Yaskawa INFORM job: A_ROOF_SIDE_0617_2_PAINT_31.JBI

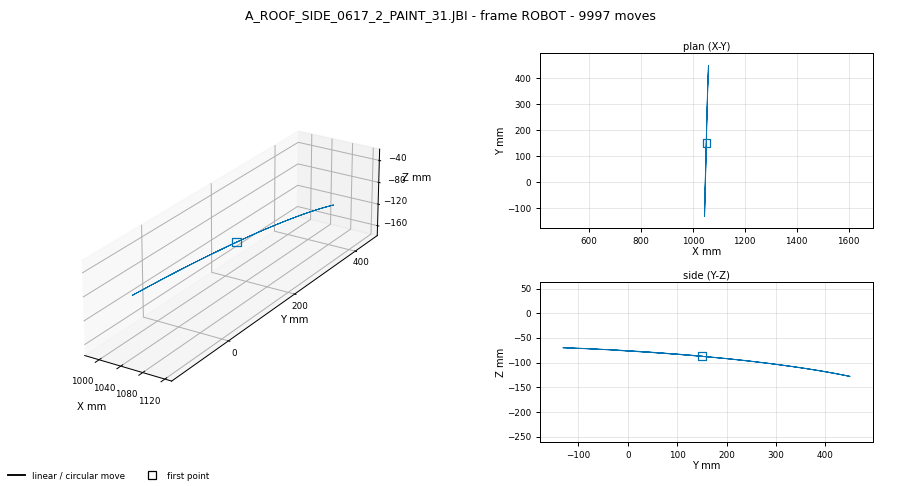
[picture p0: tool path of A_ROOF_SIDE_0617_2_PAINT_31.JBI in frame ROBOT, 9997 of 9997 moves have a stored position in this frame; points joined in program order, loops and branches not executed]
/JOB
//NAME A_ROOF_SIDE_0617_2_PAINT31
//POS
///NPOS 9997,0,0,0,0,0
///TOOL 1
///USER 0
///POSTYPE ROBOT
///RECTAN
///RCONF 1,0,0,0,0,0,0,0,0,0,0,0,0,0,0,0,0,0,0,0,0,0,0,0
C00000=1052.598,150.820,-86.690,171.369,34.301,156.430
C00001=1052.592,150.571,-86.668,171.366,34.299,156.430
C00002=1052.586,150.322,-86.647,171.364,34.297,156.430
C00003=1052.580,150.074,-86.625,171.362,34.294,156.429
C00004=1052.574,149.824,-86.603,171.360,34.291,156.429
C00005=1052.568,149.575,-86.581,171.358,34.290,156.428
C00006=1052.563,149.326,-86.560,171.357,34.287,156.428
C00007=1052.557,149.077,-86.538,171.355,34.285,156.427
C00008=1052.550,148.828,-86.516,171.353,34.283,156.427
C00009=1052.544,148.579,-86.494,171.351,34.280,156.427
C00010=1052.538,148.331,-86.473,171.349,34.278,156.426
C00011=1052.532,148.082,-86.451,171.347,34.276,156.426
C00012=1052.526,147.832,-86.429,171.345,34.273,156.425
C00013=1052.520,147.583,-86.408,171.343,34.271,156.425
C00014=1052.515,147.334,-86.386,171.341,34.269,156.425
C00015=1052.508,147.085,-86.365,171.339,34.267,156.424
C00016=1052.502,146.836,-86.343,171.337,34.264,156.424
C00017=1052.496,146.587,-86.322,171.335,34.262,156.424
C00018=1052.490,146.339,-86.300,171.334,34.260,156.423
C00019=1052.484,146.089,-86.279,171.332,34.258,156.423
C00020=1052.478,145.840,-86.257,171.330,34.255,156.422
C00021=1052.472,145.591,-86.236,171.328,34.253,156.422
C00022=1052.466,145.342,-86.214,171.326,34.251,156.422
C00023=1052.460,145.093,-86.193,171.324,34.248,156.421
C00024=1052.454,144.844,-86.171,171.322,34.246,156.421
C00025=1052.448,144.595,-86.150,171.320,34.244,156.420
C00026=1052.442,144.346,-86.128,171.318,34.242,156.420
C00027=1052.436,144.097,-86.106,171.316,34.239,156.420
C00028=1052.431,143.849,-86.085,171.314,34.237,156.419
C00029=1052.424,143.599,-86.064,171.313,34.235,156.419
C00030=1052.418,143.350,-86.042,171.311,34.233,156.418
C00031=1052.412,143.101,-86.020,171.309,34.230,156.418
C00032=1052.406,142.852,-85.999,171.307,34.228,156.418
C00033=1052.400,142.603,-85.979,171.305,34.226,156.417
C00034=1052.393,142.318,-85.954,171.303,34.223,156.417
C00035=1052.387,142.033,-85.929,171.301,34.221,156.416
C00036=1052.380,141.747,-85.905,171.298,34.218,156.416
C00037=1052.373,141.462,-85.880,171.296,34.216,156.415
C00038=1052.367,141.213,-85.858,171.294,34.213,156.415
C00039=1052.361,140.964,-85.837,171.292,34.211,156.415
C00040=1052.356,140.715,-85.816,171.291,34.209,156.414
C00041=1052.349,140.466,-85.795,171.289,34.206,156.414
C00042=1052.343,140.217,-85.774,171.287,34.204,156.413
C00043=1052.337,139.968,-85.752,171.285,34.202,156.413
C00044=1052.331,139.719,-85.731,171.284,34.200,156.413
C00045=1052.325,139.470,-85.710,171.282,34.197,156.412
C00046=1052.319,139.221,-85.689,171.280,34.195,156.412
C00047=1052.312,138.972,-85.667,171.278,34.193,156.411
C00048=1052.307,138.723,-85.646,171.275,34.191,156.411
C00049=1052.301,138.473,-85.625,171.274,34.189,156.411
C00050=1052.295,138.225,-85.604,171.272,34.187,156.410
C00051=1052.289,137.976,-85.583,171.270,34.184,156.410
C00052=1052.282,137.727,-85.561,171.268,34.182,156.410
C00053=1052.277,137.478,-85.541,171.266,34.180,156.409
C00054=1052.271,137.228,-85.519,171.265,34.178,156.409
C00055=1052.265,136.980,-85.498,171.263,34.175,156.408
C00056=1052.259,136.730,-85.478,171.261,34.173,156.408
C00057=1052.253,136.481,-85.456,171.259,34.171,156.408
C00058=1052.246,136.233,-85.435,171.258,34.169,156.407
C00059=1052.240,135.983,-85.414,171.256,34.166,156.407
C00060=1052.235,135.735,-85.393,171.254,34.164,156.406
C00061=1052.228,135.485,-85.373,171.251,34.162,156.406
C00062=1052.222,135.236,-85.351,171.249,34.160,156.406
C00063=1052.217,134.988,-85.330,171.248,34.158,156.405
C00064=1052.210,134.738,-85.309,171.246,34.155,156.405
C00065=1052.204,134.489,-85.288,171.244,34.153,156.405
C00066=1052.199,134.240,-85.267,171.242,34.151,156.404
C00067=1052.192,133.991,-85.247,171.241,34.149,156.404
C00068=1052.186,133.742,-85.226,171.239,34.146,156.403
C00069=1052.181,133.493,-85.204,171.237,34.144,156.403
C00070=1052.174,133.244,-85.183,171.235,34.142,156.403
C00071=1052.169,132.995,-85.163,171.234,34.140,156.402
C00072=1052.163,132.746,-85.141,171.232,34.137,156.402
C00073=1052.157,132.497,-85.121,171.230,34.136,156.401
C00074=1052.150,132.248,-85.100,171.227,34.133,156.401
C00075=1052.145,131.999,-85.079,171.226,34.131,156.401
C00076=1052.138,131.750,-85.058,171.224,34.129,156.400
C00077=1052.133,131.501,-85.037,171.222,34.127,156.400
C00078=1052.126,131.251,-85.017,171.220,34.125,156.400
C00079=1052.120,131.002,-84.996,171.219,34.122,156.399
C00080=1052.114,130.753,-84.976,171.217,34.120,156.399
C00081=1052.108,130.504,-84.954,171.215,34.118,156.398
C00082=1052.102,130.255,-84.934,171.213,34.116,156.398
C00083=1052.095,130.006,-84.914,171.211,34.114,156.398
C00084=1052.090,129.757,-84.892,171.210,34.111,156.397
C00085=1052.083,129.508,-84.872,171.208,34.109,156.397
C00086=1052.077,129.259,-84.851,171.206,34.107,156.397
C00087=1052.071,129.010,-84.830,171.204,34.105,156.396
C00088=1052.065,128.761,-84.810,171.203,34.103,156.396
C00089=1052.059,128.512,-84.789,171.200,34.101,156.395
C00090=1052.053,128.263,-84.769,171.198,34.098,156.395
C00091=1052.046,128.013,-84.749,171.196,34.096,156.395
C00092=1052.041,127.765,-84.727,171.195,34.095,156.394
C00093=1052.034,127.515,-84.707,171.193,34.092,156.394
C00094=1052.028,127.266,-84.687,171.191,34.090,156.394
C00095=1052.022,127.017,-84.666,171.189,34.088,156.393
C00096=1052.016,126.768,-84.645,171.188,34.086,156.393
C00097=1052.010,126.519,-84.625,171.186,34.084,156.392
C00098=1052.003,126.234,-84.601,171.184,34.081,156.392
C00099=1051.996,125.948,-84.578,171.182,34.079,156.392
C00100=1051.988,125.663,-84.554,171.180,34.076,156.391
C00101=1051.982,125.377,-84.531,171.178,34.073,156.391
C00102=1051.975,125.129,-84.511,171.176,34.071,156.390
C00103=1051.970,124.879,-84.490,171.174,34.070,156.390
C00104=1051.964,124.630,-84.470,171.172,34.067,156.390
C00105=1051.958,124.381,-84.450,171.170,34.065,156.389
C00106=1051.952,124.131,-84.429,171.168,34.063,156.389
C00107=1051.945,123.883,-84.408,171.167,34.061,156.388
C00108=1051.939,123.634,-84.388,171.165,34.059,156.388
C00109=1051.934,123.384,-84.367,171.163,34.056,156.388
C00110=1051.928,123.136,-84.347,171.162,34.054,156.387
C00111=1051.921,122.886,-84.327,171.160,34.052,156.387
C00112=1051.916,122.637,-84.306,171.158,34.050,156.387
C00113=1051.909,122.387,-84.286,171.156,34.048,156.386
C00114=1051.903,122.139,-84.265,171.155,34.046,156.386
C00115=1051.898,121.890,-84.245,171.153,34.043,156.386
C00116=1051.891,121.641,-84.224,171.151,34.041,156.385
C00117=1051.885,121.392,-84.205,171.150,34.039,156.385
C00118=1051.880,121.143,-84.184,171.147,34.037,156.384
C00119=1051.873,120.893,-84.164,171.145,34.035,156.384
C00120=1051.867,120.644,-84.144,171.143,34.032,156.384
C00121=1051.861,120.396,-84.124,171.142,34.031,156.383
C00122=1051.855,120.146,-84.103,171.140,34.028,156.383
C00123=1051.849,119.897,-84.083,171.138,34.026,156.383
C00124=1051.843,119.648,-84.063,171.137,34.024,156.382
C00125=1051.838,119.398,-84.042,171.135,34.022,156.382
C00126=1051.832,119.149,-84.022,171.133,34.020,156.381
C00127=1051.825,118.901,-84.001,171.132,34.017,156.381
C00128=1051.819,118.652,-83.981,171.130,34.015,156.381
C00129=1051.813,118.403,-83.960,171.128,34.013,156.380
C00130=1051.807,118.154,-83.941,171.126,34.011,156.380
C00131=1051.801,117.904,-83.920,171.125,34.009,156.380
C00132=1051.796,117.655,-83.900,171.123,34.006,156.379
C00133=1051.790,117.406,-83.880,171.121,34.004,156.379
C00134=1051.784,117.157,-83.860,171.119,34.002,156.378
C00135=1051.777,116.907,-83.840,171.117,34.000,156.378
C00136=1051.772,116.658,-83.820,171.115,33.998,156.378
C00137=1051.766,116.409,-83.800,171.114,33.995,156.377
C00138=1051.760,116.161,-83.780,171.112,33.993,156.377
C00139=1051.753,115.911,-83.759,171.110,33.991,156.376
C00140=1051.748,115.662,-83.739,171.109,33.989,156.376
C00141=1051.742,115.413,-83.719,171.107,33.987,156.376
C00142=1051.736,115.164,-83.699,171.105,33.984,156.375
C00143=1051.730,114.915,-83.679,171.104,33.982,156.375
C00144=1051.724,114.666,-83.658,171.102,33.980,156.375
C00145=1051.718,114.417,-83.638,171.100,33.978,156.374
C00146=1051.713,114.168,-83.619,171.099,33.975,156.374
C00147=1051.706,113.918,-83.598,171.097,33.973,156.374
C00148=1051.700,113.669,-83.578,171.095,33.971,156.373
C00149=1051.695,113.420,-83.558,171.094,33.969,156.373
C00150=1051.689,113.171,-83.538,171.092,33.967,156.372
C00151=1051.683,112.921,-83.518,171.089,33.965,156.372
C00152=1051.677,112.672,-83.498,171.088,33.963,156.372
C00153=1051.671,112.424,-83.478,171.086,33.961,156.371
C00154=1051.665,112.175,-83.458,171.084,33.959,156.371
C00155=1051.658,111.925,-83.439,171.083,33.956,156.371
C00156=1051.652,111.676,-83.419,171.081,33.954,156.370
C00157=1051.646,111.427,-83.399,171.079,33.952,156.370
C00158=1051.640,111.178,-83.379,171.078,33.950,156.369
C00159=1051.634,110.928,-83.359,171.076,33.948,156.369
C00160=1051.627,110.679,-83.340,171.074,33.946,156.369
C00161=1051.621,110.431,-83.320,171.072,33.944,156.368
C00162=1051.615,110.145,-83.297,171.071,33.941,156.368
C00163=1051.607,109.859,-83.275,171.069,33.939,156.368
C00164=1051.601,109.574,-83.252,171.067,33.936,156.367
C00165=1051.594,109.288,-83.230,171.065,33.934,156.367
C00166=1051.588,109.039,-83.210,171.063,33.932,156.366
C00167=1051.581,108.790,-83.190,171.061,33.930,156.366
C00168=1051.575,108.540,-83.170,171.059,33.928,156.366
C00169=1051.569,108.292,-83.151,171.057,33.926,156.365
C00170=1051.563,108.042,-83.132,171.055,33.923,156.365
C00171=1051.557,107.793,-83.112,171.054,33.921,156.365
C00172=1051.550,107.544,-83.091,171.052,33.919,156.364
C00173=1051.545,107.294,-83.072,171.050,33.917,156.364
C00174=1051.539,107.046,-83.052,171.049,33.915,156.364
C00175=1051.532,106.797,-83.034,171.047,33.913,156.363
C00176=1051.526,106.548,-83.014,171.045,33.911,156.363
C00177=1051.520,106.298,-82.993,171.044,33.908,156.362
C00178=1051.514,106.049,-82.974,171.042,33.906,156.362
C00179=1051.508,105.800,-82.954,171.040,33.905,156.362
C00180=1051.502,105.551,-82.935,171.039,33.903,156.361
C00181=1051.495,105.302,-82.915,171.037,33.900,156.361
C00182=1051.490,105.053,-82.896,171.035,33.898,156.361
C00183=1051.484,104.804,-82.876,171.034,33.896,156.360
C00184=1051.478,104.554,-82.857,171.032,33.894,156.360
C00185=1051.472,104.305,-82.837,171.030,33.892,156.360
C00186=1051.466,104.055,-82.817,171.029,33.890,156.359
C00187=1051.459,103.807,-82.798,171.027,33.888,156.359
C00188=1051.453,103.557,-82.779,171.025,33.885,156.359
C00189=1051.447,103.309,-82.759,171.023,33.883,156.358
C00190=1051.442,103.059,-82.740,171.021,33.881,156.358
C00191=1051.436,102.810,-82.720,171.020,33.879,156.357
C00192=1051.429,102.561,-82.701,171.018,33.877,156.357
C00193=1051.423,102.311,-82.681,171.016,33.875,156.357
C00194=1051.417,102.062,-82.661,171.015,33.872,156.356
C00195=1051.411,101.813,-82.642,171.013,33.870,156.356
C00196=1051.405,101.564,-82.622,171.011,33.868,156.356
C00197=1051.399,101.315,-82.604,171.010,33.866,156.355
C00198=1051.393,101.066,-82.584,171.008,33.864,156.355
C00199=1051.387,100.817,-82.564,171.006,33.862,156.355
C00200=1051.382,100.567,-82.545,171.005,33.860,156.354
C00201=1051.375,100.318,-82.527,171.003,33.857,156.354
C00202=1051.369,100.069,-82.507,171.001,33.856,156.353
C00203=1051.363,99.820,-82.488,171.000,33.854,156.353
C00204=1051.356,99.570,-82.468,170.998,33.852,156.353
C00205=1051.350,99.321,-82.448,170.996,33.850,156.353
C00206=1051.344,99.072,-82.430,170.995,33.847,156.352
C00207=1051.338,98.823,-82.410,170.993,33.845,156.352
C00208=1051.332,98.574,-82.391,170.991,33.843,156.351
C00209=1051.326,98.325,-82.372,170.989,33.841,156.351
C00210=1051.319,98.076,-82.353,170.987,33.839,156.351
C00211=1051.314,97.826,-82.334,170.986,33.837,156.350
C00212=1051.307,97.578,-82.315,170.984,33.835,156.350
C00213=1051.301,97.328,-82.295,170.982,33.833,156.350
C00214=1051.296,97.079,-82.276,170.981,33.831,156.349
C00215=1051.289,96.830,-82.257,170.979,33.829,156.349
C00216=1051.284,96.580,-82.238,170.977,33.826,156.349
C00217=1051.277,96.332,-82.219,170.976,33.825,156.348
C00218=1051.271,96.082,-82.199,170.974,33.823,156.348
C00219=1051.264,95.833,-82.181,170.972,33.821,156.348
C00220=1051.258,95.583,-82.161,170.971,33.818,156.347
C00221=1051.252,95.334,-82.143,170.969,33.816,156.347
C00222=1051.246,95.085,-82.123,170.968,33.814,156.347
C00223=1051.240,94.836,-82.104,170.966,33.812,156.346
C00224=1051.234,94.587,-82.085,170.964,33.810,156.346
C00225=1051.227,94.338,-82.066,170.963,33.808,156.345
C00226=1051.221,94.053,-82.044,170.961,33.806,156.345
C00227=1051.213,93.766,-82.023,170.959,33.803,156.345
C00228=1051.207,93.481,-82.001,170.957,33.801,156.344
C00229=1051.200,93.196,-81.979,170.954,33.798,156.344
C00230=1051.194,92.946,-81.960,170.953,33.796,156.343
C00231=1051.188,92.697,-81.941,170.951,33.794,156.343
C00232=1051.182,92.448,-81.922,170.949,33.792,156.343
C00233=1051.176,92.199,-81.903,170.948,33.790,156.342
C00234=1051.170,91.950,-81.884,170.946,33.788,156.342
C00235=1051.163,91.701,-81.865,170.944,33.786,156.342
C00236=1051.158,91.451,-81.846,170.943,33.784,156.341
C00237=1051.151,91.202,-81.827,170.941,33.781,156.341
C00238=1051.146,90.953,-81.808,170.939,33.779,156.341
C00239=1051.140,90.703,-81.789,170.938,33.777,156.340
C00240=1051.134,90.454,-81.770,170.936,33.775,156.340
C00241=1051.127,90.205,-81.751,170.935,33.773,156.340
C00242=1051.121,89.955,-81.732,170.933,33.771,156.339
C00243=1051.115,89.706,-81.713,170.931,33.769,156.339
C00244=1051.109,89.457,-81.695,170.930,33.767,156.339
C00245=1051.102,89.208,-81.676,170.928,33.765,156.338
C00246=1051.096,88.959,-81.657,170.926,33.763,156.338
C00247=1051.090,88.710,-81.638,170.925,33.761,156.338
C00248=1051.084,88.460,-81.620,170.923,33.759,156.337
C00249=1051.077,88.211,-81.602,170.921,33.756,156.337
C00250=1051.072,87.961,-81.582,170.920,33.755,156.337
C00251=1051.065,87.712,-81.564,170.918,33.753,156.336
C00252=1051.059,87.463,-81.545,170.917,33.751,156.336
C00253=1051.053,87.215,-81.527,170.915,33.749,156.336
C00254=1051.047,86.965,-81.508,170.913,33.747,156.335
C00255=1051.041,86.716,-81.489,170.911,33.745,156.335
C00256=1051.035,86.467,-81.470,170.909,33.742,156.335
C00257=1051.028,86.217,-81.452,170.907,33.740,156.334
C00258=1051.022,85.968,-81.434,170.906,33.738,156.334
C00259=1051.016,85.719,-81.414,170.904,33.736,156.334
C00260=1051.010,85.469,-81.396,170.903,33.734,156.333
C00261=1051.004,85.220,-81.377,170.901,33.732,156.333
C00262=1050.997,84.971,-81.359,170.899,33.730,156.333
C00263=1050.992,84.721,-81.340,170.898,33.728,156.332
C00264=1050.986,84.473,-81.322,170.896,33.726,156.332
C00265=1050.979,84.224,-81.303,170.894,33.724,156.331
C00266=1050.973,83.975,-81.284,170.893,33.722,156.331
C00267=1050.967,83.725,-81.266,170.891,33.720,156.331
C00268=1050.961,83.475,-81.247,170.890,33.718,156.331
C00269=1050.955,83.226,-81.229,170.888,33.716,156.330
C00270=1050.948,82.977,-81.210,170.886,33.714,156.330
C00271=1050.943,82.729,-81.192,170.885,33.712,156.329
C00272=1050.937,82.479,-81.173,170.883,33.710,156.329
C00273=1050.931,82.230,-81.154,170.881,33.708,156.329
C00274=1050.924,81.980,-81.136,170.880,33.705,156.328
C00275=1050.918,81.731,-81.118,170.878,33.703,156.328
C00276=1050.912,81.482,-81.099,170.877,33.701,156.328
C00277=1050.907,81.233,-81.080,170.875,33.699,156.327
C00278=1050.900,80.984,-81.062,170.873,33.697,156.327
C00279=1050.894,80.734,-81.044,170.872,33.695,156.327
C00280=1050.888,80.485,-81.025,170.870,33.693,156.326
C00281=1050.881,80.236,-81.006,170.868,33.691,156.326
C00282=1050.876,79.987,-80.989,170.866,33.689,156.326
C00283=1050.870,79.737,-80.970,170.864,33.687,156.325
C00284=1050.864,79.488,-80.951,170.863,33.685,156.325
C00285=1050.858,79.238,-80.933,170.861,33.682,156.325
C00286=1050.851,78.989,-80.914,170.859,33.680,156.324
C00287=1050.846,78.740,-80.897,170.858,33.679,156.324
C00288=1050.839,78.491,-80.878,170.856,33.677,156.324
C00289=1050.833,78.242,-80.860,170.855,33.675,156.323
C00290=1050.826,77.956,-80.838,170.853,33.672,156.323
C00291=1050.819,77.670,-80.818,170.851,33.670,156.323
C00292=1050.812,77.384,-80.797,170.849,33.667,156.322
C00293=1050.805,77.099,-80.776,170.847,33.665,156.322
C00294=1050.798,76.850,-80.757,170.845,33.663,156.321
C00295=1050.793,76.601,-80.740,170.844,33.661,156.321
C00296=1050.786,76.352,-80.721,170.842,33.659,156.321
C00297=1050.780,76.102,-80.703,170.841,33.657,156.320
C00298=1050.774,75.853,-80.685,170.839,33.655,156.320
C00299=1050.768,75.603,-80.667,170.837,33.653,156.320
C00300=1050.762,75.354,-80.648,170.836,33.651,156.319
C00301=1050.756,75.105,-80.630,170.834,33.649,156.319
C00302=1050.749,74.856,-80.612,170.832,33.647,156.319
C00303=1050.743,74.606,-80.594,170.831,33.645,156.318
C00304=1050.737,74.357,-80.576,170.829,33.643,156.318
C00305=1050.731,74.108,-80.558,170.828,33.641,156.318
C00306=1050.725,73.859,-80.539,170.826,33.639,156.317
C00307=1050.718,73.609,-80.522,170.824,33.637,156.317
C00308=1050.713,73.360,-80.504,170.823,33.635,156.317
C00309=1050.706,73.111,-80.485,170.821,33.633,156.316
C00310=1050.700,72.861,-80.468,170.820,33.631,156.316
C00311=1050.694,72.612,-80.449,170.818,33.629,156.316
C00312=1050.688,72.363,-80.431,170.816,33.626,156.315
C00313=1050.682,72.113,-80.413,170.814,33.624,156.315
C00314=1050.676,71.864,-80.395,170.812,33.622,156.315
C00315=1050.670,71.615,-80.377,170.810,33.620,156.314
C00316=1050.664,71.366,-80.359,170.809,33.619,156.314
C00317=1050.657,71.117,-80.341,170.807,33.617,156.314
C00318=1050.651,70.867,-80.323,170.806,33.615,156.313
C00319=1050.645,70.618,-80.305,170.804,33.613,156.313
C00320=1050.639,70.369,-80.287,170.802,33.611,156.313
C00321=1050.633,70.119,-80.269,170.801,33.608,156.312
C00322=1050.627,69.871,-80.251,170.799,33.606,156.312
C00323=1050.621,69.621,-80.233,170.797,33.604,156.312
C00324=1050.614,69.371,-80.216,170.796,33.602,156.311
C00325=1050.608,69.122,-80.198,170.794,33.600,156.311
C00326=1050.602,68.873,-80.179,170.793,33.598,156.311
C00327=1050.596,68.623,-80.161,170.791,33.596,156.310
C00328=1050.590,68.374,-80.144,170.789,33.594,156.310
C00329=1050.583,68.125,-80.126,170.788,33.592,156.310
C00330=1050.577,67.876,-80.108,170.786,33.590,156.309
C00331=1050.571,67.627,-80.090,170.784,33.588,156.309
C00332=1050.565,67.377,-80.072,170.783,33.586,156.309
C00333=1050.558,67.128,-80.055,170.781,33.584,156.309
C00334=1050.553,66.879,-80.037,170.780,33.582,156.308
C00335=1050.546,66.630,-80.019,170.778,33.580,156.308
C00336=1050.540,66.380,-80.001,170.776,33.578,156.307
C00337=1050.534,66.131,-79.984,170.775,33.576,156.307
C00338=1050.528,65.881,-79.966,170.773,33.574,156.307
C00339=1050.521,65.632,-79.949,170.771,33.572,156.306
C00340=1050.515,65.383,-79.930,170.770,33.570,156.306
C00341=1050.509,65.134,-79.912,170.768,33.568,156.306
C00342=1050.503,64.884,-79.894,170.767,33.566,156.306
C00343=1050.497,64.635,-79.877,170.765,33.564,156.305
C00344=1050.491,64.386,-79.860,170.763,33.562,156.305
C00345=1050.485,64.136,-79.842,170.762,33.560,156.305
C00346=1050.478,63.887,-79.825,170.760,33.558,156.304
C00347=1050.472,63.637,-79.807,170.758,33.556,156.304
C00348=1050.466,63.389,-79.790,170.757,33.554,156.304
C00349=1050.459,63.140,-79.772,170.755,33.552,156.303
C00350=1050.453,62.890,-79.754,170.753,33.550,156.303
C00351=1050.446,62.641,-79.737,170.752,33.548,156.303
C00352=1050.440,62.392,-79.719,170.750,33.546,156.302
C00353=1050.433,62.142,-79.702,170.749,33.545,156.302
C00354=1050.426,61.856,-79.682,170.746,33.543,156.302
C00355=1050.419,61.570,-79.662,170.744,33.541,156.301
C00356=1050.412,61.284,-79.642,170.742,33.538,156.301
C00357=1050.405,60.999,-79.622,170.740,33.536,156.301
C00358=1050.399,60.749,-79.604,170.738,33.534,156.300
C00359=1050.392,60.500,-79.587,170.737,33.532,156.300
C00360=1050.386,60.251,-79.569,170.735,33.530,156.300
C00361=1050.379,60.001,-79.552,170.733,33.528,156.299
C00362=1050.374,59.752,-79.535,170.732,33.526,156.299
C00363=1050.367,59.503,-79.517,170.730,33.524,156.299
C00364=1050.361,59.254,-79.500,170.729,33.522,156.298
C00365=1050.355,59.004,-79.482,170.727,33.520,156.298
C00366=1050.348,58.755,-79.465,170.725,33.518,156.298
C00367=1050.342,58.506,-79.447,170.724,33.516,156.297
C00368=1050.335,58.256,-79.430,170.722,33.514,156.297
C00369=1050.329,58.008,-79.413,170.720,33.513,156.297
C00370=1050.323,57.758,-79.395,170.719,33.511,156.297
C00371=1050.317,57.509,-79.378,170.717,33.509,156.296
C00372=1050.311,57.259,-79.361,170.715,33.507,156.296
C00373=1050.305,57.010,-79.344,170.714,33.505,156.296
C00374=1050.298,56.761,-79.327,170.712,33.503,156.295
C00375=1050.292,56.511,-79.309,170.711,33.501,156.295
C00376=1050.285,56.262,-79.292,170.709,33.499,156.295
C00377=1050.279,56.012,-79.274,170.707,33.497,156.294
C00378=1050.273,55.763,-79.258,170.706,33.495,156.294
C00379=1050.267,55.514,-79.240,170.704,33.493,156.294
C00380=1050.261,55.264,-79.223,170.702,33.491,156.293
C00381=1050.254,55.015,-79.205,170.701,33.489,156.293
C00382=1050.249,54.766,-79.188,170.699,33.487,156.293
C00383=1050.242,54.516,-79.171,170.697,33.485,156.293
C00384=1050.236,54.267,-79.154,170.696,33.483,156.292
C00385=1050.230,54.017,-79.136,170.694,33.481,156.292
C00386=1050.223,53.769,-79.119,170.692,33.479,156.292
C00387=1050.217,53.519,-79.102,170.691,33.477,156.291
C00388=1050.211,53.270,-79.085,170.689,33.475,156.291
C00389=1050.205,53.020,-79.068,170.688,33.473,156.291
C00390=1050.199,52.771,-79.050,170.686,33.471,156.290
C00391=1050.193,52.522,-79.033,170.684,33.469,156.290
C00392=1050.186,52.272,-79.017,170.683,33.467,156.290
C00393=1050.181,52.023,-78.999,170.681,33.465,156.289
C00394=1050.174,51.774,-78.982,170.679,33.463,156.289
C00395=1050.168,51.525,-78.965,170.678,33.462,156.289
C00396=1050.162,51.275,-78.947,170.676,33.459,156.288
C00397=1050.155,51.026,-78.931,170.674,33.457,156.288
C00398=1050.149,50.776,-78.914,170.673,33.456,156.288
C00399=1050.143,50.527,-78.896,170.671,33.454,156.287
C00400=1050.137,50.278,-78.879,170.670,33.452,156.287
C00401=1050.131,50.028,-78.863,170.668,33.450,156.287
C00402=1050.125,49.779,-78.845,170.666,33.448,156.287
C00403=1050.118,49.530,-78.828,170.665,33.446,156.286
C00404=1050.113,49.280,-78.811,170.663,33.444,156.286
C00405=1050.107,49.031,-78.794,170.661,33.442,156.286
C00406=1050.100,48.782,-78.777,170.660,33.440,156.285
C00407=1050.095,48.532,-78.760,170.658,33.438,156.285
C00408=1050.088,48.283,-78.742,170.657,33.436,156.285
C00409=1050.082,48.034,-78.726,170.655,33.434,156.284
C00410=1050.076,47.785,-78.709,170.653,33.432,156.284
C00411=1050.069,47.535,-78.691,170.652,33.430,156.284
C00412=1050.064,47.286,-78.675,170.650,33.428,156.283
C00413=1050.057,47.037,-78.658,170.648,33.426,156.283
C00414=1050.051,46.787,-78.641,170.647,33.424,156.283
C00415=1050.045,46.538,-78.624,170.644,33.422,156.282
C00416=1050.039,46.289,-78.608,170.642,33.420,156.282
C00417=1050.033,46.039,-78.590,170.641,33.418,156.282
C00418=1050.026,45.752,-78.570,170.639,33.415,156.281
C00419=1050.019,45.467,-78.551,170.637,33.413,156.281
C00420=1050.012,45.180,-78.532,170.635,33.411,156.281
C00421=1050.005,44.894,-78.512,170.633,33.409,156.280
C00422=1049.999,44.645,-78.496,170.632,33.407,156.280
C00423=1049.993,44.396,-78.479,170.630,33.405,156.280
C00424=1049.988,44.146,-78.462,170.628,33.403,156.279
C00425=1049.981,43.897,-78.445,170.627,33.401,156.279
C00426=1049.975,43.648,-78.428,170.625,33.399,156.279
C00427=1049.969,43.399,-78.411,170.623,33.397,156.278
C00428=1049.963,43.149,-78.394,170.622,33.395,156.278
C00429=1049.957,42.900,-78.377,170.620,33.393,156.278
C00430=1049.951,42.650,-78.361,170.619,33.391,156.277
C00431=1049.944,42.400,-78.344,170.617,33.389,156.277
C00432=1049.938,42.152,-78.327,170.615,33.387,156.277
C00433=1049.932,41.902,-78.311,170.614,33.386,156.277
C00434=1049.925,41.652,-78.294,170.612,33.384,156.276
C00435=1049.919,41.404,-78.277,170.610,33.382,156.276
C00436=1049.913,41.154,-78.261,170.609,33.380,156.276
C00437=1049.906,40.905,-78.244,170.607,33.378,156.275
C00438=1049.900,40.655,-78.228,170.605,33.376,156.275
C00439=1049.894,40.406,-78.211,170.604,33.374,156.275
C00440=1049.888,40.157,-78.194,170.602,33.372,156.274
C00441=1049.882,39.907,-78.178,170.600,33.370,156.274
C00442=1049.876,39.658,-78.161,170.599,33.368,156.274
C00443=1049.870,39.409,-78.145,170.597,33.366,156.273
C00444=1049.863,39.159,-78.128,170.595,33.364,156.273
C00445=1049.858,38.910,-78.111,170.594,33.362,156.273
C00446=1049.852,38.660,-78.095,170.592,33.360,156.273
C00447=1049.845,38.411,-78.078,170.590,33.358,156.272
C00448=1049.839,38.161,-78.061,170.589,33.356,156.272
C00449=1049.833,37.912,-78.045,170.587,33.354,156.272
C00450=1049.827,37.663,-78.029,170.585,33.352,156.271
C00451=1049.821,37.414,-78.012,170.584,33.350,156.271
C00452=1049.813,37.164,-77.996,170.582,33.348,156.271
C00453=1049.807,36.915,-77.979,170.580,33.347,156.271
C00454=1049.801,36.666,-77.963,170.579,33.345,156.270
C00455=1049.795,36.415,-77.946,170.577,33.343,156.270
C00456=1049.789,36.166,-77.930,170.575,33.341,156.270
C00457=1049.783,35.917,-77.913,170.574,33.339,156.269
C00458=1049.777,35.668,-77.897,170.572,33.338,156.269
C00459=1049.769,35.418,-77.881,170.570,33.336,156.269
C00460=1049.764,35.169,-77.865,170.569,33.334,156.268
C00461=1049.758,34.920,-77.848,170.567,33.332,156.268
C00462=1049.752,34.670,-77.832,170.565,33.330,156.268
C00463=1049.745,34.421,-77.815,170.564,33.328,156.268
C00464=1049.739,34.171,-77.799,170.562,33.326,156.267
C00465=1049.732,33.922,-77.783,170.560,33.324,156.267
C00466=1049.726,33.673,-77.767,170.558,33.322,156.267
C00467=1049.720,33.424,-77.750,170.557,33.320,156.266
C00468=1049.714,33.174,-77.734,170.555,33.318,156.266
C00469=1049.708,32.924,-77.718,170.553,33.317,156.266
C00470=1049.701,32.675,-77.702,170.552,33.315,156.266
C00471=1049.695,32.426,-77.686,170.550,33.313,156.265
C00472=1049.689,32.177,-77.669,170.548,33.311,156.265
C00473=1049.683,31.927,-77.653,170.547,33.309,156.265
C00474=1049.677,31.677,-77.636,170.545,33.307,156.264
C00475=1049.671,31.428,-77.620,170.543,33.306,156.264
C00476=1049.664,31.179,-77.605,170.542,33.304,156.264
C00477=1049.658,30.929,-77.588,170.540,33.302,156.264
C00478=1049.651,30.679,-77.572,170.538,33.300,156.263
C00479=1049.646,30.430,-77.555,170.537,33.298,156.263
C00480=1049.640,30.181,-77.539,170.535,33.296,156.263
C00481=1049.633,29.932,-77.524,170.533,33.294,156.262
C00482=1049.625,29.645,-77.505,170.531,33.292,156.262
C00483=1049.619,29.360,-77.486,170.529,33.290,156.262
C00484=1049.612,29.073,-77.467,170.527,33.288,156.261
C00485=1049.605,28.787,-77.449,170.526,33.286,156.261
C00486=1049.599,28.538,-77.432,170.524,33.284,156.261
C00487=1049.592,28.289,-77.417,170.522,33.282,156.260
C00488=1049.586,28.039,-77.401,170.520,33.280,156.260
C00489=1049.580,27.790,-77.384,170.519,33.278,156.260
C00490=1049.573,27.540,-77.369,170.517,33.276,156.260
C00491=1049.567,27.290,-77.353,170.515,33.274,156.259
C00492=1049.560,27.041,-77.337,170.514,33.272,156.259
C00493=1049.555,26.792,-77.321,170.512,33.271,156.259
C00494=1049.549,26.543,-77.305,170.510,33.269,156.258
C00495=1049.542,26.294,-77.289,170.509,33.267,156.258
C00496=1049.536,26.044,-77.273,170.507,33.265,156.258
C00497=1049.530,25.794,-77.257,170.505,33.263,156.258
C00498=1049.523,25.545,-77.241,170.503,33.261,156.257
C00499=1049.517,25.295,-77.225,170.502,33.259,156.257
C00500=1049.510,25.046,-77.209,170.500,33.257,156.257
C00501=1049.504,24.797,-77.193,170.498,33.256,156.257
C00502=1049.498,24.548,-77.177,170.497,33.254,156.256
C00503=1049.492,24.298,-77.162,170.495,33.252,156.256
C00504=1049.486,24.048,-77.145,170.493,33.251,156.256
C00505=1049.479,23.799,-77.130,170.491,33.249,156.255
C00506=1049.473,23.550,-77.114,170.490,33.247,156.255
C00507=1049.466,23.300,-77.098,170.488,33.245,156.255
C00508=1049.461,23.050,-77.082,170.486,33.243,156.255
C00509=1049.454,22.801,-77.066,170.485,33.241,156.254
C00510=1049.448,22.552,-77.050,170.483,33.239,156.254
C00511=1049.442,22.302,-77.035,170.481,33.237,156.254
C00512=1049.436,22.053,-77.019,170.480,33.236,156.253
C00513=1049.430,21.804,-77.003,170.478,33.234,156.253
C00514=1049.423,21.554,-76.988,170.476,33.232,156.253
C00515=1049.417,21.305,-76.971,170.474,33.230,156.253
C00516=1049.411,21.056,-76.956,170.473,33.228,156.252
C00517=1049.405,20.806,-76.940,170.471,33.226,156.252
C00518=1049.398,20.557,-76.925,170.469,33.224,156.252
C00519=1049.392,20.307,-76.908,170.468,33.223,156.252
C00520=1049.386,20.058,-76.893,170.466,33.221,156.251
C00521=1049.380,19.808,-76.877,170.464,33.219,156.251
C00522=1049.373,19.559,-76.861,170.462,33.218,156.251
C00523=1049.368,19.309,-76.846,170.461,33.216,156.250
C00524=1049.361,19.060,-76.830,170.459,33.214,156.250
C00525=1049.355,18.811,-76.814,170.457,33.212,156.250
C00526=1049.349,18.561,-76.799,170.455,33.210,156.250
C00527=1049.342,18.312,-76.783,170.454,33.208,156.249
C00528=1049.336,18.062,-76.768,170.452,33.207,156.249
C00529=1049.330,17.813,-76.752,170.450,33.205,156.249
C00530=1049.324,17.563,-76.737,170.449,33.203,156.248
C00531=1049.317,17.314,-76.721,170.447,33.201,156.248
C00532=1049.311,17.064,-76.706,170.445,33.199,156.248
C00533=1049.305,16.815,-76.690,170.443,33.197,156.248
C00534=1049.298,16.566,-76.674,170.442,33.196,156.247
C00535=1049.293,16.316,-76.659,170.440,33.194,156.247
C00536=1049.286,16.067,-76.643,170.438,33.192,156.247
C00537=1049.280,15.817,-76.628,170.436,33.191,156.247
C00538=1049.274,15.568,-76.612,170.435,33.189,156.246
C00539=1049.267,15.318,-76.597,170.433,33.187,156.246
C00540=1049.261,15.069,-76.580,170.431,33.185,156.246
C00541=1049.255,14.819,-76.565,170.429,33.183,156.246
C00542=1049.248,14.570,-76.550,170.428,33.181,156.245
C00543=1049.243,14.320,-76.534,170.426,33.180,156.245
C00544=1049.236,14.071,-76.519,170.424,33.178,156.245
C00545=1049.229,13.822,-76.504,170.422,33.176,156.244
C00546=1049.224,13.605,-76.491,170.421,33.174,156.244
C00547=1049.218,13.389,-76.477,170.419,33.173,156.244
C00548=1049.213,13.173,-76.464,170.418,33.172,156.244
C00549=1049.208,12.957,-76.450,170.416,33.170,156.244
C00550=1049.202,12.740,-76.437,170.415,33.168,156.243
C00551=1049.196,12.524,-76.424,170.413,33.167,156.243
C00552=1049.191,12.307,-76.411,170.412,33.166,156.243
C00553=1049.185,12.091,-76.397,170.410,33.164,156.243
C00554=1049.179,11.842,-76.382,170.408,33.162,156.242
C00555=1049.173,11.592,-76.367,170.407,33.161,156.242
C00556=1049.166,11.343,-76.352,170.405,33.159,156.242
C00557=1049.160,11.093,-76.336,170.403,33.157,156.242
C00558=1049.154,10.843,-76.321,170.401,33.155,156.241
C00559=1049.147,10.594,-76.306,170.400,33.154,156.241
C00560=1049.141,10.345,-76.291,170.398,33.152,156.241
C00561=1049.135,10.096,-76.276,170.397,33.150,156.241
C00562=1049.129,9.846,-76.261,170.395,33.148,156.240
C00563=1049.122,9.597,-76.245,170.394,33.147,156.240
C00564=1049.116,9.347,-76.230,170.392,33.145,156.240
C00565=1049.110,9.097,-76.215,170.390,33.143,156.240
C00566=1049.103,8.848,-76.199,170.388,33.142,156.239
C00567=1049.097,8.599,-76.184,170.386,33.140,156.239
C00568=1049.090,8.349,-76.169,170.385,33.138,156.239
C00569=1049.084,8.099,-76.154,170.383,33.136,156.239
C00570=1049.077,7.850,-76.139,170.381,33.135,156.238
C00571=1049.072,7.601,-76.124,170.379,33.133,156.238
C00572=1049.066,7.351,-76.109,170.378,33.131,156.238
C00573=1049.060,7.102,-76.094,170.376,33.129,156.238
C00574=1049.051,6.751,-76.072,170.373,33.127,156.237
C00575=1049.042,6.399,-76.051,170.371,33.125,156.237
C00576=1049.033,6.049,-76.030,170.368,33.122,156.237
C00577=1049.024,5.697,-76.009,170.366,33.120,156.236
C00578=1049.018,5.447,-75.994,170.364,33.118,156.236
C00579=1049.011,5.198,-75.978,170.362,33.116,156.236
C00580=1049.005,4.949,-75.963,170.360,33.114,156.235
C00581=1048.999,4.699,-75.948,170.359,33.113,156.235
C00582=1048.993,4.450,-75.934,170.357,33.111,156.235
C00583=1048.986,4.200,-75.919,170.355,33.109,156.235
C00584=1048.980,3.951,-75.904,170.353,33.107,156.234
C00585=1048.974,3.701,-75.889,170.352,33.106,156.234
C00586=1048.967,3.451,-75.874,170.350,33.104,156.234
C00587=1048.961,3.203,-75.859,170.348,33.103,156.234
C00588=1048.955,2.953,-75.843,170.346,33.101,156.233
C00589=1048.949,2.703,-75.828,170.344,33.099,156.233
C00590=1048.943,2.454,-75.813,170.343,33.097,156.233
C00591=1048.937,2.205,-75.799,170.341,33.096,156.233
C00592=1048.931,1.955,-75.784,170.339,33.094,156.232
C00593=1048.924,1.706,-75.769,170.337,33.092,156.232
C00594=1048.918,1.456,-75.754,170.335,33.090,156.232
C00595=1048.912,1.207,-75.739,170.334,33.088,156.232
C00596=1048.906,0.957,-75.724,170.332,33.087,156.231
C00597=1048.899,0.708,-75.709,170.330,33.085,156.231
C00598=1048.893,0.458,-75.694,170.328,33.083,156.231
C00599=1048.887,0.209,-75.680,170.326,33.081,156.231
C00600=1048.881,-0.041,-75.665,170.325,33.080,156.230
C00601=1048.874,-0.290,-75.650,170.323,33.078,156.230
C00602=1048.869,-0.539,-75.635,170.321,33.077,156.230
C00603=1048.862,-0.789,-75.620,170.319,33.075,156.230
C00604=1048.857,-1.039,-75.605,170.317,33.073,156.229
C00605=1048.850,-1.289,-75.590,170.316,33.071,156.229
C00606=1048.844,-1.537,-75.575,170.314,33.070,156.229
C00607=1048.838,-1.787,-75.560,170.312,33.068,156.229
C00608=1048.832,-2.037,-75.546,170.310,33.066,156.228
C00609=1048.826,-2.286,-75.531,170.308,33.064,156.228
C00610=1048.819,-2.569,-75.515,170.306,33.062,156.228
C00611=1048.811,-2.852,-75.498,170.304,33.060,156.228
C00612=1048.805,-3.135,-75.482,170.302,33.059,156.227
C00613=1048.797,-3.418,-75.464,170.300,33.057,156.227
C00614=1048.791,-3.667,-75.450,170.298,33.055,156.227
C00615=1048.785,-3.918,-75.435,170.297,33.053,156.227
C00616=1048.779,-4.167,-75.421,170.295,33.052,156.226
C00617=1048.772,-4.416,-75.406,170.293,33.050,156.226
C00618=1048.766,-4.666,-75.391,170.291,33.048,156.226
C00619=1048.760,-4.915,-75.377,170.289,33.047,156.226
C00620=1048.754,-5.164,-75.362,170.287,33.045,156.225
C00621=1048.747,-5.414,-75.348,170.286,33.044,156.225
C00622=1048.741,-5.663,-75.334,170.284,33.042,156.225
C00623=1048.735,-5.913,-75.319,170.283,33.040,156.225
C00624=1048.728,-6.162,-75.304,170.281,33.039,156.225
C00625=1048.721,-6.412,-75.290,170.279,33.037,156.224
C00626=1048.716,-6.661,-75.276,170.277,33.035,156.224
C00627=1048.709,-6.911,-75.261,170.276,33.034,156.224
C00628=1048.702,-7.160,-75.246,170.274,33.032,156.224
C00629=1048.697,-7.410,-75.232,170.272,33.030,156.223
C00630=1048.690,-7.660,-75.217,170.270,33.029,156.223
C00631=1048.684,-7.909,-75.203,170.268,33.028,156.223
C00632=1048.678,-8.158,-75.189,170.266,33.025,156.223
C00633=1048.671,-8.408,-75.174,170.264,33.024,156.222
C00634=1048.665,-8.657,-75.160,170.263,33.023,156.222
C00635=1048.659,-8.907,-75.146,170.261,33.021,156.222
C00636=1048.652,-9.157,-75.131,170.259,33.019,156.222
C00637=1048.646,-9.406,-75.117,170.257,33.018,156.222
C00638=1048.640,-9.656,-75.102,170.255,33.016,156.221
C00639=1048.634,-9.905,-75.088,170.253,33.014,156.221
C00640=1048.628,-10.154,-75.073,170.252,33.013,156.221
C00641=1048.621,-10.405,-75.059,170.250,33.012,156.221
C00642=1048.615,-10.653,-75.045,170.248,33.009,156.220
C00643=1048.609,-10.903,-75.031,170.246,33.008,156.220
C00644=1048.603,-11.152,-75.016,170.244,33.007,156.220
C00645=1048.596,-11.402,-75.002,170.242,33.005,156.220
C00646=1048.590,-11.652,-74.988,170.240,33.003,156.220
C00647=1048.584,-11.901,-74.973,170.239,33.002,156.219
C00648=1048.577,-12.151,-74.960,170.237,33.000,156.219
C00649=1048.571,-12.400,-74.945,170.235,32.998,156.219
C00650=1048.565,-12.650,-74.931,170.233,32.997,156.219
C00651=1048.559,-12.899,-74.917,170.231,32.995,156.218
C00652=1048.552,-13.148,-74.902,170.229,32.993,156.218
C00653=1048.547,-13.398,-74.888,170.227,32.992,156.218
C00654=1048.541,-13.648,-74.873,170.225,32.991,156.218
C00655=1048.534,-13.897,-74.860,170.224,32.989,156.218
C00656=1048.528,-14.147,-74.845,170.222,32.987,156.217
C00657=1048.522,-14.396,-74.832,170.220,32.986,156.217
C00658=1048.515,-14.646,-74.817,170.218,32.984,156.217
C00659=1048.509,-14.896,-74.802,170.216,32.982,156.217
C00660=1048.503,-15.144,-74.788,170.214,32.981,156.216
C00661=1048.497,-15.395,-74.774,170.212,32.979,156.216
C00662=1048.491,-15.644,-74.761,170.210,32.977,156.216
C00663=1048.484,-15.894,-74.746,170.209,32.976,156.216
C00664=1048.478,-16.143,-74.733,170.207,32.975,156.216
C00665=1048.472,-16.393,-74.718,170.205,32.973,156.215
C00666=1048.465,-16.642,-74.704,170.203,32.972,156.215
C00667=1048.459,-16.892,-74.690,170.202,32.970,156.215
C00668=1048.453,-17.141,-74.676,170.200,32.968,156.215
C00669=1048.447,-17.391,-74.662,170.198,32.967,156.215
C00670=1048.440,-17.640,-74.648,170.196,32.965,156.214
C00671=1048.433,-17.890,-74.634,170.194,32.964,156.214
C00672=1048.428,-18.139,-74.621,170.193,32.962,156.214
C00673=1048.421,-18.389,-74.606,170.191,32.961,156.214
C00674=1048.414,-18.670,-74.591,170.188,32.959,156.214
C00675=1048.407,-18.951,-74.575,170.186,32.957,156.213
C00676=1048.400,-19.233,-74.559,170.184,32.955,156.213
C00677=1048.393,-19.514,-74.544,170.182,32.954,156.213
C00678=1048.387,-19.764,-74.530,170.180,32.953,156.213
C00679=1048.380,-20.013,-74.515,170.178,32.951,156.213
C00680=1048.374,-20.263,-74.502,170.176,32.950,156.212
C00681=1048.368,-20.513,-74.488,170.174,32.948,156.212
C00682=1048.362,-20.762,-74.475,170.172,32.946,156.212
C00683=1048.355,-21.011,-74.460,170.171,32.945,156.212
C00684=1048.349,-21.261,-74.446,170.169,32.943,156.211
C00685=1048.342,-21.511,-74.433,170.167,32.942,156.211
C00686=1048.337,-21.761,-74.419,170.165,32.941,156.211
C00687=1048.330,-22.009,-74.405,170.163,32.939,156.211
C00688=1048.323,-22.259,-74.391,170.161,32.937,156.211
C00689=1048.318,-22.509,-74.377,170.159,32.936,156.210
C00690=1048.311,-22.759,-74.364,170.157,32.934,156.210
C00691=1048.306,-23.008,-74.350,170.155,32.933,156.210
C00692=1048.299,-23.257,-74.336,170.153,32.931,156.210
C00693=1048.292,-23.507,-74.322,170.151,32.930,156.210
C00694=1048.287,-23.756,-74.308,170.149,32.928,156.210
C00695=1048.280,-24.006,-74.295,170.148,32.927,156.209
C00696=1048.274,-24.256,-74.281,170.146,32.925,156.209
C00697=1048.268,-24.505,-74.268,170.144,32.924,156.209
C00698=1048.261,-24.755,-74.253,170.142,32.922,156.209
C00699=1048.256,-25.004,-74.239,170.140,32.921,156.208
C00700=1048.250,-25.253,-74.226,170.138,32.919,156.208
C00701=1048.243,-25.503,-74.212,170.136,32.918,156.208
C00702=1048.237,-25.753,-74.199,170.134,32.916,156.208
C00703=1048.231,-26.002,-74.185,170.133,32.915,156.208
C00704=1048.224,-26.252,-74.172,170.131,32.913,156.208
C00705=1048.219,-26.502,-74.158,170.129,32.912,156.207
C00706=1048.213,-26.751,-74.145,170.127,32.910,156.207
C00707=1048.205,-27.000,-74.130,170.125,32.909,156.207
C00708=1048.200,-27.250,-74.116,170.123,32.907,156.207
C00709=1048.193,-27.500,-74.103,170.121,32.906,156.207
C00710=1048.187,-27.749,-74.089,170.120,32.904,156.206
C00711=1048.181,-27.998,-74.076,170.118,32.903,156.206
C00712=1048.174,-28.248,-74.063,170.116,32.902,156.206
C00713=1048.168,-28.498,-74.049,170.114,32.901,156.206
C00714=1048.161,-28.747,-74.036,170.112,32.899,156.206
C00715=1048.155,-28.997,-74.022,170.110,32.898,156.206
C00716=1048.149,-29.247,-74.009,170.108,32.896,156.205
C00717=1048.143,-29.496,-73.996,170.106,32.895,156.205
C00718=1048.136,-29.746,-73.982,170.104,32.893,156.205
C00719=1048.130,-29.996,-73.969,170.102,32.892,156.205
C00720=1048.124,-30.245,-73.956,170.100,32.890,156.205
C00721=1048.117,-30.495,-73.942,170.098,32.889,156.204
C00722=1048.111,-30.744,-73.929,170.096,32.888,156.204
C00723=1048.105,-30.993,-73.916,170.094,32.886,156.204
C00724=1048.099,-31.244,-73.901,170.092,32.885,156.204
C00725=1048.092,-31.493,-73.888,170.090,32.883,156.204
C00726=1048.086,-31.742,-73.875,170.088,32.882,156.203
C00727=1048.080,-31.991,-73.862,170.086,32.880,156.203
C00728=1048.074,-32.242,-73.849,170.084,32.880,156.203
C00729=1048.067,-32.491,-73.835,170.082,32.878,156.203
C00730=1048.061,-32.741,-73.822,170.080,32.877,156.203
C00731=1048.055,-32.990,-73.809,170.078,32.875,156.203
C00732=1048.048,-33.240,-73.795,170.076,32.874,156.203
C00733=1048.042,-33.489,-73.782,170.074,32.872,156.202
C00734=1048.036,-33.738,-73.769,170.072,32.871,156.202
C00735=1048.030,-33.989,-73.756,170.071,32.869,156.202
C00736=1048.024,-34.238,-73.742,170.069,32.868,156.202
C00737=1048.017,-34.488,-73.729,170.067,32.867,156.202
C00738=1048.010,-34.768,-73.714,170.065,32.865,156.201
C00739=1048.003,-35.049,-73.699,170.063,32.864,156.201
C00740=1047.997,-35.330,-73.684,170.061,32.862,156.201
C00741=1047.990,-35.610,-73.669,170.058,32.861,156.201
C00742=1047.983,-35.859,-73.656,170.056,32.859,156.201
C00743=1047.977,-36.110,-73.643,170.054,32.858,156.201
C00744=1047.971,-36.359,-73.630,170.053,32.856,156.200
C00745=1047.964,-36.608,-73.617,170.051,32.855,156.200
C00746=1047.958,-36.857,-73.603,170.049,32.854,156.200
C00747=1047.952,-37.107,-73.591,170.047,32.852,156.200
C00748=1047.946,-37.357,-73.577,170.045,32.851,156.200
C00749=1047.939,-37.606,-73.564,170.043,32.850,156.200
C00750=1047.933,-37.856,-73.551,170.041,32.848,156.199
C00751=1047.927,-38.106,-73.538,170.039,32.847,156.199
C00752=1047.921,-38.355,-73.525,170.037,32.845,156.199
C00753=1047.915,-38.605,-73.512,170.035,32.844,156.199
C00754=1047.909,-38.854,-73.499,170.033,32.843,156.199
C00755=1047.902,-39.104,-73.485,170.031,32.842,156.199
C00756=1047.896,-39.354,-73.473,170.029,32.840,156.198
C00757=1047.890,-39.603,-73.459,170.027,32.839,156.198
C00758=1047.884,-39.852,-73.446,170.024,32.837,156.198
C00759=1047.877,-40.102,-73.434,170.022,32.837,156.198
C00760=1047.871,-40.351,-73.421,170.020,32.835,156.198
C00761=1047.864,-40.602,-73.408,170.018,32.834,156.198
C00762=1047.858,-40.851,-73.395,170.016,32.832,156.197
C00763=1047.852,-41.101,-73.382,170.014,32.831,156.197
C00764=1047.846,-41.350,-73.369,170.013,32.830,156.197
C00765=1047.839,-41.600,-73.357,170.011,32.828,156.197
C00766=1047.833,-41.849,-73.344,170.009,32.828,156.197
C00767=1047.827,-42.098,-73.330,170.007,32.826,156.197
C00768=1047.820,-42.349,-73.318,170.005,32.825,156.197
C00769=1047.814,-42.598,-73.304,170.003,32.823,156.196
C00770=1047.808,-42.848,-73.292,170.001,32.822,156.196
C00771=1047.801,-43.097,-73.279,169.999,32.821,156.196
C00772=1047.795,-43.347,-73.266,169.997,32.820,156.196
C00773=1047.789,-43.596,-73.253,169.995,32.819,156.196
C00774=1047.783,-43.846,-73.241,169.993,32.817,156.196
C00775=1047.777,-44.096,-73.229,169.991,32.816,156.195
C00776=1047.770,-44.345,-73.215,169.989,32.815,156.195
C00777=1047.765,-44.595,-73.203,169.987,32.814,156.195
C00778=1047.758,-44.845,-73.189,169.985,32.812,156.195
C00779=1047.752,-45.095,-73.177,169.983,32.811,156.195
C00780=1047.745,-45.344,-73.164,169.981,32.810,156.195
C00781=1047.739,-45.593,-73.151,169.979,32.808,156.195
C00782=1047.733,-45.843,-73.139,169.977,32.808,156.195
C00783=1047.727,-46.093,-73.126,169.975,32.806,156.194
C00784=1047.721,-46.342,-73.113,169.973,32.805,156.194
C00785=1047.714,-46.591,-73.100,169.971,32.803,156.194
C00786=1047.708,-46.841,-73.088,169.969,32.802,156.194
C00787=1047.702,-47.091,-73.075,169.967,32.801,156.194
C00788=1047.696,-47.340,-73.062,169.964,32.800,156.194
C00789=1047.689,-47.590,-73.050,169.962,32.799,156.194
C00790=1047.683,-47.840,-73.037,169.960,32.797,156.193
C00791=1047.677,-48.089,-73.024,169.959,32.796,156.193
C00792=1047.671,-48.339,-73.012,169.957,32.795,156.193
C00793=1047.665,-48.589,-73.000,169.955,32.793,156.193
C00794=1047.658,-48.838,-72.986,169.953,32.793,156.193
C00795=1047.652,-49.088,-72.974,169.951,32.791,156.193
C00796=1047.647,-49.338,-72.961,169.949,32.790,156.193
C00797=1047.640,-49.587,-72.949,169.947,32.789,156.192
C00798=1047.634,-49.837,-72.936,169.945,32.787,156.192
C00799=1047.628,-50.086,-72.924,169.943,32.786,156.192
C00800=1047.622,-50.336,-72.911,169.941,32.785,156.192
C00801=1047.615,-50.586,-72.899,169.939,32.784,156.192
C00802=1047.608,-50.867,-72.885,169.936,32.783,156.192
C00803=1047.601,-51.148,-72.871,169.934,32.781,156.192
C00804=1047.594,-51.428,-72.857,169.932,32.780,156.192
C00805=1047.586,-51.710,-72.843,169.929,32.779,156.191
C00806=1047.580,-51.959,-72.831,169.927,32.778,156.191
C00807=1047.574,-52.209,-72.818,169.925,32.777,156.191
C00808=1047.567,-52.459,-72.806,169.923,32.776,156.191
C00809=1047.561,-52.709,-72.794,169.921,32.774,156.191
C00810=1047.554,-52.958,-72.781,169.919,32.773,156.191
C00811=1047.548,-53.207,-72.769,169.917,32.773,156.191
C00812=1047.542,-53.457,-72.756,169.915,32.771,156.191
C00813=1047.535,-53.707,-72.744,169.913,32.770,156.191
C00814=1047.529,-53.957,-72.732,169.910,32.769,156.190
C00815=1047.523,-54.205,-72.720,169.908,32.768,156.190
C00816=1047.516,-54.455,-72.708,169.906,32.767,156.190
C00817=1047.511,-54.705,-72.696,169.905,32.766,156.190
C00818=1047.504,-54.954,-72.684,169.903,32.765,156.190
C00819=1047.498,-55.204,-72.671,169.901,32.764,156.190
C00820=1047.491,-55.454,-72.659,169.899,32.763,156.190
C00821=1047.485,-55.703,-72.647,169.897,32.762,156.190
C00822=1047.479,-55.953,-72.635,169.895,32.760,156.189
C00823=1047.472,-56.203,-72.623,169.893,32.759,156.189
C00824=1047.466,-56.452,-72.610,169.890,32.758,156.189
C00825=1047.459,-56.702,-72.598,169.888,32.757,156.189
C00826=1047.453,-56.951,-72.586,169.886,32.756,156.189
C00827=1047.447,-57.201,-72.573,169.884,32.755,156.189
C00828=1047.440,-57.451,-72.562,169.882,32.754,156.189
C00829=1047.434,-57.700,-72.550,169.880,32.753,156.189
C00830=1047.428,-57.950,-72.538,169.878,32.752,156.189
C00831=1047.422,-58.200,-72.526,169.876,32.751,156.189
C00832=1047.416,-58.450,-72.513,169.873,32.750,156.188
C00833=1047.409,-58.699,-72.501,169.871,32.749,156.188
C00834=1047.403,-58.949,-72.489,169.869,32.748,156.188
C00835=1047.397,-59.199,-72.477,169.867,32.747,156.188
C00836=1047.391,-59.448,-72.465,169.865,32.746,156.188
C00837=1047.384,-59.697,-72.453,169.863,32.744,156.188
C00838=1047.378,-59.947,-72.441,169.861,32.744,156.188
C00839=1047.371,-60.197,-72.429,169.859,32.743,156.188
C00840=1047.365,-60.446,-72.417,169.857,32.741,156.188
C00841=1047.359,-60.696,-72.404,169.854,32.740,156.188
C00842=1047.353,-60.946,-72.393,169.853,32.740,156.188
C00843=1047.346,-61.195,-72.381,169.851,32.739,156.187
C00844=1047.341,-61.445,-72.369,169.849,32.737,156.187
C00845=1047.334,-61.695,-72.357,169.847,32.736,156.187
C00846=1047.327,-61.944,-72.345,169.845,32.736,156.187
C00847=1047.322,-62.193,-72.333,169.843,32.734,156.187
C00848=1047.316,-62.443,-72.321,169.841,32.733,156.187
C00849=1047.309,-62.693,-72.309,169.838,32.732,156.187
C00850=1047.303,-62.943,-72.297,169.836,32.732,156.187
C00851=1047.296,-63.193,-72.285,169.834,32.730,156.187
C00852=1047.290,-63.441,-72.273,169.832,32.729,156.187
C00853=1047.285,-63.692,-72.262,169.830,32.728,156.186
C00854=1047.278,-63.941,-72.250,169.828,32.727,156.186
C00855=1047.271,-64.191,-72.238,169.826,32.726,156.186
C00856=1047.266,-64.440,-72.225,169.823,32.725,156.186
C00857=1047.260,-64.690,-72.213,169.821,32.724,156.186
C00858=1047.253,-64.940,-72.202,169.819,32.723,156.186
C00859=1047.247,-65.190,-72.190,169.817,32.722,156.186
C00860=1047.241,-65.439,-72.178,169.815,32.721,156.186
C00861=1047.235,-65.689,-72.167,169.813,32.720,156.186
C00862=1047.228,-65.938,-72.155,169.811,32.719,156.186
C00863=1047.223,-66.188,-72.143,169.808,32.718,156.186
C00864=1047.216,-66.437,-72.131,169.806,32.717,156.185
C00865=1047.210,-66.687,-72.119,169.804,32.716,156.185
C00866=1047.203,-66.969,-72.106,169.803,32.715,156.185
C00867=1047.196,-67.252,-72.093,169.800,32.714,156.185
C00868=1047.189,-67.534,-72.079,169.798,32.713,156.185
C00869=1047.182,-67.817,-72.066,169.795,32.712,156.185
C00870=1047.176,-68.066,-72.054,169.793,32.711,156.185
C00871=1047.170,-68.316,-72.043,169.791,32.710,156.185
C00872=1047.164,-68.566,-72.031,169.789,32.709,156.185
C00873=1047.158,-68.815,-72.019,169.787,32.708,156.185
C00874=1047.152,-69.065,-72.008,169.785,32.707,156.184
C00875=1047.145,-69.314,-71.996,169.783,32.706,156.184
C00876=1047.140,-69.564,-71.984,169.780,32.705,156.184
C00877=1047.133,-69.814,-71.972,169.778,32.704,156.184
C00878=1047.127,-70.063,-71.960,169.776,32.703,156.184
C00879=1047.122,-70.313,-71.949,169.774,32.702,156.184
C00880=1047.115,-70.563,-71.937,169.772,32.701,156.184
C00881=1047.109,-70.812,-71.926,169.770,32.700,156.184
C00882=1047.103,-71.062,-71.914,169.768,32.699,156.184
C00883=1047.097,-71.312,-71.902,169.765,32.698,156.184
C00884=1047.091,-71.561,-71.891,169.763,32.698,156.184
C00885=1047.085,-71.811,-71.880,169.761,32.696,156.184
C00886=1047.079,-72.060,-71.868,169.759,32.695,156.184
C00887=1047.072,-72.310,-71.857,169.757,32.694,156.183
C00888=1047.066,-72.560,-71.844,169.755,32.694,156.183
C00889=1047.061,-72.810,-71.833,169.753,32.693,156.183
C00890=1047.054,-73.059,-71.821,169.751,32.692,156.183
C00891=1047.048,-73.309,-71.810,169.749,32.691,156.183
C00892=1047.042,-73.559,-71.798,169.747,32.690,156.183
C00893=1047.037,-73.808,-71.787,169.745,32.689,156.183
C00894=1047.030,-74.058,-71.775,169.743,32.688,156.183
C00895=1047.024,-74.307,-71.764,169.740,32.687,156.183
C00896=1047.018,-74.557,-71.752,169.738,32.686,156.183
C00897=1047.011,-74.807,-71.741,169.736,32.685,156.183
C00898=1047.006,-75.057,-71.730,169.734,32.684,156.183
C00899=1046.999,-75.306,-71.718,169.732,32.684,156.183
C00900=1046.993,-75.556,-71.707,169.729,32.683,156.183
C00901=1046.987,-75.806,-71.696,169.727,32.682,156.183
C00902=1046.981,-76.055,-71.684,169.725,32.682,156.183
C00903=1046.974,-76.305,-71.673,169.723,32.681,156.182
C00904=1046.968,-76.555,-71.662,169.721,32.680,156.182
C00905=1046.962,-76.804,-71.650,169.718,32.679,156.182
C00906=1046.956,-77.054,-71.639,169.716,32.678,156.182
C00907=1046.950,-77.304,-71.628,169.714,32.677,156.182
C00908=1046.943,-77.553,-71.616,169.712,32.676,156.182
C00909=1046.938,-77.803,-71.605,169.710,32.676,156.182
C00910=1046.931,-78.053,-71.594,169.707,32.675,156.182
C00911=1046.925,-78.302,-71.584,169.705,32.674,156.182
C00912=1046.918,-78.552,-71.572,169.703,32.673,156.182
C00913=1046.912,-78.801,-71.561,169.702,32.673,156.182
C00914=1046.906,-79.051,-71.550,169.700,32.672,156.182
C00915=1046.900,-79.301,-71.539,169.697,32.671,156.182
C00916=1046.894,-79.550,-71.527,169.695,32.670,156.182
C00917=1046.888,-79.800,-71.516,169.693,32.669,156.182
C00918=1046.882,-80.050,-71.505,169.691,32.669,156.182
C00919=1046.876,-80.300,-71.494,169.689,32.668,156.182
C00920=1046.869,-80.549,-71.483,169.686,32.667,156.182
C00921=1046.863,-80.798,-71.472,169.684,32.667,156.182
C00922=1046.856,-81.049,-71.460,169.682,32.666,156.182
C00923=1046.851,-81.298,-71.450,169.680,32.666,156.182
C00924=1046.844,-81.548,-71.439,169.677,32.665,156.182
C00925=1046.838,-81.797,-71.428,169.675,32.664,156.181
C00926=1046.831,-82.048,-71.417,169.673,32.663,156.181
C00927=1046.825,-82.297,-71.407,169.671,32.663,156.181
C00928=1046.819,-82.547,-71.395,169.668,32.662,156.181
C00929=1046.813,-82.796,-71.384,169.666,32.661,156.181
C00930=1046.805,-83.081,-71.371,169.664,32.661,156.181
C00931=1046.798,-83.365,-71.359,169.661,32.660,156.181
C00932=1046.792,-83.650,-71.347,169.659,32.659,156.181
C00933=1046.784,-83.935,-71.334,169.656,32.658,156.181
C00934=1046.777,-84.184,-71.324,169.654,32.658,156.181
C00935=1046.771,-84.434,-71.312,169.652,32.657,156.181
C00936=1046.765,-84.683,-71.301,169.650,32.656,156.181
C00937=1046.759,-84.933,-71.291,169.648,32.656,156.181
C00938=1046.752,-85.183,-71.280,169.646,32.655,156.181
C00939=1046.747,-85.432,-71.269,169.644,32.654,156.181
C00940=1046.740,-85.682,-71.258,169.641,32.654,156.181
C00941=1046.734,-85.932,-71.247,169.639,32.653,156.181
C00942=1046.728,-86.181,-71.237,169.637,32.652,156.181
C00943=1046.722,-86.431,-71.225,169.635,32.652,156.181
C00944=1046.715,-86.680,-71.215,169.632,32.651,156.181
C00945=1046.709,-86.931,-71.204,169.630,32.650,156.181
C00946=1046.703,-87.180,-71.193,169.628,32.650,156.181
C00947=1046.697,-87.429,-71.183,169.626,32.649,156.181
C00948=1046.690,-87.680,-71.171,169.623,32.649,156.181
C00949=1046.685,-87.929,-71.161,169.621,32.648,156.181
C00950=1046.678,-88.179,-71.150,169.619,32.647,156.181
C00951=1046.672,-88.429,-71.140,169.617,32.647,156.181
C00952=1046.666,-88.678,-71.129,169.614,32.646,156.181
C00953=1046.659,-88.928,-71.118,169.612,32.646,156.181
C00954=1046.654,-89.178,-71.107,169.610,32.645,156.181
C00955=1046.647,-89.427,-71.097,169.608,32.644,156.181
C00956=1046.641,-89.677,-71.086,169.605,32.644,156.181
C00957=1046.635,-89.927,-71.075,169.603,32.643,156.181
C00958=1046.629,-90.176,-71.065,169.601,32.643,156.181
C00959=1046.623,-90.427,-71.054,169.600,32.642,156.181
C00960=1046.617,-90.676,-71.043,169.597,32.642,156.181
C00961=1046.610,-90.925,-71.033,169.595,32.641,156.181
C00962=1046.605,-91.175,-71.022,169.593,32.640,156.181
C00963=1046.598,-91.425,-71.011,169.591,32.640,156.181
C00964=1046.592,-91.674,-71.001,169.588,32.639,156.181
C00965=1046.586,-91.924,-70.990,169.586,32.638,156.181
C00966=1046.579,-92.174,-70.980,169.584,32.638,156.181
C00967=1046.574,-92.424,-70.969,169.582,32.637,156.181
C00968=1046.568,-92.673,-70.958,169.579,32.636,156.181
C00969=1046.562,-92.923,-70.948,169.577,32.636,156.181
C00970=1046.555,-93.173,-70.937,169.575,32.635,156.181
C00971=1046.549,-93.422,-70.927,169.573,32.635,156.181
C00972=1046.543,-93.672,-70.916,169.570,32.634,156.181
C00973=1046.538,-93.922,-70.906,169.568,32.634,156.181
C00974=1046.531,-94.172,-70.895,169.566,32.633,156.181
C00975=1046.525,-94.421,-70.884,169.563,32.633,156.181
C00976=1046.518,-94.671,-70.874,169.561,32.632,156.181
C00977=1046.513,-94.921,-70.864,169.559,32.632,156.181
C00978=1046.507,-95.170,-70.853,169.557,32.631,156.181
C00979=1046.500,-95.420,-70.842,169.554,32.631,156.181
C00980=1046.495,-95.670,-70.832,169.552,32.630,156.181
C00981=1046.488,-95.919,-70.822,169.550,32.630,156.181
C00982=1046.482,-96.169,-70.811,169.549,32.629,156.181
C00983=1046.477,-96.419,-70.801,169.546,32.629,156.181
C00984=1046.470,-96.669,-70.790,169.544,32.628,156.181
C00985=1046.464,-96.918,-70.779,169.542,32.627,156.181
C00986=1046.458,-97.168,-70.770,169.540,32.627,156.181
C00987=1046.452,-97.418,-70.759,169.537,32.626,156.181
C00988=1046.446,-97.667,-70.749,169.535,32.626,156.181
C00989=1046.440,-97.918,-70.738,169.533,32.625,156.181
C00990=1046.434,-98.167,-70.729,169.530,32.625,156.181
C00991=1046.427,-98.417,-70.718,169.528,32.625,156.181
C00992=1046.421,-98.666,-70.707,169.526,32.624,156.181
C00993=1046.415,-98.916,-70.698,169.524,32.624,156.181
C00994=1046.408,-99.202,-70.686,169.521,32.623,156.181
C00995=1046.401,-99.490,-70.674,169.518,32.623,156.181
C00996=1046.394,-99.776,-70.662,169.516,32.622,156.181
C00997=1046.386,-100.063,-70.650,169.513,32.622,156.181
C00998=1046.380,-100.313,-70.641,169.511,32.622,156.181
C00999=1046.375,-100.562,-70.630,169.508,32.621,156.181
C01000=1046.368,-100.812,-70.620,169.506,32.621,156.181
C01001=1046.361,-101.062,-70.610,169.504,32.620,156.181
C01002=1046.356,-101.312,-70.600,169.501,32.620,156.181
C01003=1046.350,-101.562,-70.590,169.499,32.619,156.181
C01004=1046.343,-101.811,-70.580,169.498,32.619,156.181
C01005=1046.338,-102.061,-70.570,169.496,32.619,156.181
C01006=1046.331,-102.310,-70.559,169.493,32.618,156.181
C01007=1046.325,-102.560,-70.550,169.491,32.618,156.181
C01008=1046.319,-102.809,-70.539,169.489,32.617,156.181
C01009=1046.313,-103.060,-70.529,169.486,32.617,156.181
C01010=1046.306,-103.310,-70.519,169.484,32.617,156.181
C01011=1046.301,-103.559,-70.509,169.482,32.617,156.181
C01012=1046.295,-103.809,-70.499,169.479,32.616,156.181
C01013=1046.288,-104.059,-70.489,169.477,32.615,156.181
C01014=1046.282,-104.308,-70.479,169.475,32.615,156.181
C01015=1046.276,-104.558,-70.469,169.473,32.615,156.181
C01016=1046.270,-104.807,-70.459,169.470,32.615,156.181
C01017=1046.264,-105.057,-70.449,169.468,32.615,156.182
C01018=1046.258,-105.307,-70.439,169.466,32.614,156.182
C01019=1046.252,-105.557,-70.429,169.463,32.614,156.182
C01020=1046.246,-105.806,-70.419,169.461,32.613,156.182
C01021=1046.240,-106.056,-70.410,169.459,32.613,156.182
C01022=1046.234,-106.306,-70.399,169.456,32.613,156.182
C01023=1046.228,-106.555,-70.389,169.454,32.612,156.182
C01024=1046.221,-106.806,-70.379,169.452,32.612,156.182
C01025=1046.215,-107.056,-70.370,169.449,32.612,156.182
C01026=1046.208,-107.305,-70.360,169.447,32.612,156.182
C01027=1046.203,-107.555,-70.349,169.445,32.611,156.182
C01028=1046.197,-107.805,-70.340,169.443,32.611,156.182
C01029=1046.190,-108.054,-70.330,169.441,32.611,156.182
C01030=1046.184,-108.304,-70.320,169.439,32.611,156.182
C01031=1046.178,-108.553,-70.310,169.436,32.610,156.182
C01032=1046.172,-108.803,-70.301,169.434,32.610,156.182
C01033=1046.165,-109.053,-70.291,169.432,32.610,156.182
C01034=1046.159,-109.303,-70.281,169.429,32.610,156.182
C01035=1046.154,-109.553,-70.271,169.427,32.609,156.182
C01036=1046.148,-109.803,-70.262,169.425,32.609,156.182
C01037=1046.141,-110.052,-70.251,169.423,32.609,156.183
C01038=1046.135,-110.302,-70.242,169.420,32.609,156.183
C01039=1046.129,-110.551,-70.232,169.418,32.609,156.183
C01040=1046.123,-110.801,-70.223,169.416,32.608,156.183
C01041=1046.116,-111.051,-70.213,169.413,32.608,156.183
C01042=1046.110,-111.301,-70.204,169.411,32.608,156.183
C01043=1046.104,-111.551,-70.194,169.409,32.608,156.183
C01044=1046.098,-111.800,-70.184,169.406,32.607,156.183
C01045=1046.092,-112.050,-70.175,169.404,32.607,156.183
C01046=1046.086,-112.299,-70.165,169.402,32.607,156.183
C01047=1046.080,-112.549,-70.155,169.399,32.607,156.183
C01048=1046.074,-112.799,-70.145,169.397,32.607,156.183
C01049=1046.068,-113.048,-70.136,169.395,32.607,156.183
C01050=1046.062,-113.298,-70.126,169.392,32.606,156.183
C01051=1046.056,-113.548,-70.117,169.391,32.606,156.183
C01052=1046.050,-113.798,-70.107,169.389,32.606,156.183
C01053=1046.043,-114.048,-70.097,169.386,32.606,156.183
C01054=1046.037,-114.297,-70.088,169.384,32.606,156.184
C01055=1046.031,-114.547,-70.078,169.381,32.605,156.184
C01056=1046.025,-114.797,-70.069,169.379,32.605,156.184
C01057=1046.019,-115.047,-70.059,169.377,32.605,156.184
C01058=1046.012,-115.332,-70.049,169.374,32.605,156.184
C01059=1046.005,-115.618,-70.038,169.371,32.605,156.184
C01060=1045.998,-115.903,-70.027,169.369,32.605,156.184
C01061=1045.991,-116.190,-70.016,169.366,32.605,156.184
C01062=1045.985,-116.440,-70.007,169.364,32.605,156.184
C01063=1045.979,-116.690,-69.997,169.361,32.604,156.184
C01064=1045.973,-116.939,-69.988,169.359,32.604,156.184
C01065=1045.967,-117.188,-69.978,169.357,32.604,156.184
C01066=1045.961,-117.438,-69.969,169.354,32.604,156.185
C01067=1045.954,-117.688,-69.960,169.352,32.604,156.185
C01068=1045.948,-117.938,-69.950,169.350,32.604,156.185
C01069=1045.942,-118.187,-69.941,169.347,32.604,156.185
C01070=1045.936,-118.438,-69.932,169.345,32.604,156.185
C01071=1045.930,-118.687,-69.923,169.343,32.604,156.185
C01072=1045.924,-118.937,-69.913,169.340,32.603,156.185
C01073=1045.918,-119.186,-69.903,169.338,32.604,156.185
C01074=1045.912,-119.436,-69.894,169.336,32.604,156.185
C01075=1045.905,-119.686,-69.884,169.334,32.603,156.185
C01076=1045.899,-119.936,-69.876,169.332,32.604,156.185
C01077=1045.893,-120.185,-69.867,169.329,32.603,156.186
C01078=1045.887,-120.435,-69.857,169.327,32.603,156.186
C01079=1045.881,-120.685,-69.848,169.325,32.604,156.186
C01080=1045.875,-120.935,-69.838,169.322,32.603,156.186
C01081=1045.869,-121.185,-69.829,169.320,32.603,156.186
C01082=1045.863,-121.434,-69.820,169.318,32.604,156.186
C01083=1045.856,-121.684,-69.811,169.315,32.603,156.186
C01084=1045.850,-121.933,-69.802,169.313,32.603,156.186
C01085=1045.844,-122.184,-69.793,169.310,32.603,156.186
C01086=1045.838,-122.434,-69.783,169.308,32.603,156.186
C01087=1045.833,-122.683,-69.774,169.306,32.604,156.186
C01088=1045.827,-122.933,-69.765,169.303,32.603,156.187
C01089=1045.820,-123.183,-69.756,169.301,32.603,156.187
C01090=1045.814,-123.432,-69.747,169.299,32.603,156.187
C01091=1045.808,-123.682,-69.737,169.296,32.603,156.187
C01092=1045.802,-123.932,-69.728,169.294,32.604,156.187
C01093=1045.796,-124.182,-69.719,169.292,32.603,156.187
C01094=1045.789,-124.431,-69.710,169.289,32.603,156.187
C01095=1045.784,-124.681,-69.701,169.287,32.603,156.187
C01096=1045.778,-124.931,-69.692,169.284,32.603,156.187
C01097=1045.772,-125.181,-69.683,169.282,32.604,156.187
C01098=1045.765,-125.431,-69.674,169.280,32.603,156.188
C01099=1045.759,-125.680,-69.665,169.278,32.604,156.188
C01100=1045.753,-125.930,-69.656,169.276,32.604,156.188
C01101=1045.747,-126.180,-69.647,169.274,32.604,156.188
C01102=1045.741,-126.430,-69.638,169.271,32.604,156.188
C01103=1045.735,-126.679,-69.629,169.269,32.604,156.188
C01104=1045.728,-126.929,-69.620,169.266,32.604,156.188
C01105=1045.722,-127.179,-69.611,169.264,32.604,156.188
C01106=1045.717,-127.428,-69.602,169.262,32.605,156.189
C01107=1045.710,-127.678,-69.594,169.259,32.604,156.189
C01108=1045.705,-127.927,-69.584,169.257,32.605,156.189
C01109=1045.699,-128.177,-69.574,169.255,32.604,156.189
C01110=1045.696,-128.428,-69.563,169.253,32.603,156.189
C01111=1045.693,-128.677,-69.553,169.251,32.602,156.188
C01112=1045.690,-128.927,-69.541,169.249,32.599,156.188
C01113=1045.689,-129.177,-69.529,169.247,32.597,156.188
C01114=1045.689,-129.428,-69.516,169.245,32.595,156.188
C01115=1045.690,-129.679,-69.503,169.244,32.591,156.187
C01116=1045.692,-129.928,-69.489,169.242,32.587,156.186
C01117=1045.695,-130.178,-69.474,169.241,32.583,156.186
C01118=1045.699,-130.429,-69.459,169.240,32.579,156.185
C01119=1045.703,-130.680,-69.443,169.240,32.574,156.184
C01120=1045.708,-130.930,-69.426,169.239,32.568,156.183
C01121=1045.714,-131.179,-69.409,169.238,32.562,156.182
C01122=1045.358,-131.203,-69.650,169.192,32.741,156.215
C01123=1045.352,-130.953,-69.667,169.192,32.747,156.216
C01124=1045.346,-130.703,-69.683,169.193,32.752,156.217
C01125=1045.342,-130.453,-69.699,169.194,32.757,156.217
C01126=1045.338,-130.202,-69.714,169.196,32.762,156.218
C01127=1045.335,-129.952,-69.729,169.197,32.767,156.219
C01128=1045.333,-129.702,-69.744,169.198,32.770,156.219
C01129=1045.333,-129.451,-69.757,169.200,32.773,156.220
C01130=1045.333,-129.201,-69.770,169.201,32.777,156.220
C01131=1045.334,-128.951,-69.782,169.202,32.779,156.221
C01132=1045.336,-128.701,-69.794,169.204,32.781,156.221
C01133=1045.339,-128.451,-69.805,169.206,32.782,156.221
C01134=1045.343,-128.202,-69.815,169.208,32.783,156.221
C01135=1045.348,-127.951,-69.824,169.210,32.783,156.221
C01136=1045.354,-127.702,-69.834,169.213,32.784,156.221
C01137=1045.359,-127.453,-69.843,169.215,32.783,156.221
C01138=1045.365,-127.202,-69.852,169.218,32.784,156.221
C01139=1045.372,-126.953,-69.861,169.220,32.783,156.221
C01140=1045.377,-126.703,-69.870,169.222,32.783,156.221
C01141=1045.384,-126.453,-69.879,169.225,32.783,156.221
C01142=1045.391,-126.204,-69.888,169.227,32.783,156.220
C01143=1045.396,-125.954,-69.897,169.229,32.783,156.220
C01144=1045.402,-125.704,-69.906,169.232,32.783,156.220
C01145=1045.409,-125.454,-69.914,169.234,32.783,156.220
C01146=1045.415,-125.204,-69.924,169.237,32.782,156.220
C01147=1045.420,-124.955,-69.933,169.239,32.782,156.220
C01148=1045.426,-124.705,-69.942,169.241,32.782,156.220
C01149=1045.433,-124.455,-69.951,169.244,32.782,156.220
C01150=1045.439,-124.205,-69.961,169.246,32.782,156.219
C01151=1045.445,-123.956,-69.969,169.249,32.782,156.219
C01152=1045.451,-123.706,-69.979,169.251,32.782,156.219
C01153=1045.458,-123.456,-69.988,169.253,32.782,156.219
C01154=1045.463,-123.206,-69.996,169.256,32.782,156.219
C01155=1045.469,-122.957,-70.006,169.258,32.782,156.219
C01156=1045.475,-122.707,-70.015,169.259,32.782,156.219
C01157=1045.481,-122.457,-70.024,169.262,32.782,156.219
C01158=1045.487,-122.207,-70.034,169.264,32.782,156.219
C01159=1045.494,-121.958,-70.042,169.267,32.782,156.219
C01160=1045.500,-121.708,-70.052,169.269,32.782,156.219
C01161=1045.506,-121.458,-70.061,169.271,32.782,156.218
C01162=1045.512,-121.208,-70.070,169.274,32.782,156.218
C01163=1045.518,-120.958,-70.080,169.276,32.782,156.218
C01164=1045.524,-120.709,-70.089,169.278,32.782,156.218
C01165=1045.530,-120.459,-70.097,169.281,32.782,156.218
C01166=1045.536,-120.209,-70.107,169.283,32.782,156.218
C01167=1045.542,-119.960,-70.116,169.286,32.782,156.218
C01168=1045.549,-119.710,-70.126,169.288,32.782,156.218
C01169=1045.554,-119.461,-70.135,169.290,32.782,156.218
C01170=1045.560,-119.210,-70.144,169.293,32.782,156.218
C01171=1045.566,-118.960,-70.154,169.295,32.782,156.217
C01172=1045.572,-118.711,-70.163,169.297,32.782,156.217
C01173=1045.579,-118.461,-70.173,169.300,32.782,156.217
C01174=1045.585,-118.211,-70.182,169.302,32.782,156.217
C01175=1045.591,-117.962,-70.191,169.304,32.782,156.217
C01176=1045.597,-117.712,-70.200,169.307,32.782,156.217
C01177=1045.603,-117.462,-70.209,169.309,32.782,156.217
C01178=1045.609,-117.212,-70.219,169.312,32.782,156.217
C01179=1045.615,-116.962,-70.228,169.314,32.782,156.217
C01180=1045.622,-116.713,-70.238,169.316,32.783,156.217
C01181=1045.628,-116.463,-70.248,169.318,32.782,156.217
C01182=1045.633,-116.214,-70.257,169.320,32.782,156.217
C01183=1045.641,-115.927,-70.267,169.323,32.783,156.217
C01184=1045.648,-115.641,-70.279,169.325,32.783,156.216
C01185=1045.655,-115.357,-70.289,169.328,32.783,156.216
C01186=1045.662,-115.070,-70.300,169.331,32.783,156.216
C01187=1045.668,-114.820,-70.310,169.333,32.783,156.216
C01188=1045.674,-114.570,-70.319,169.336,32.783,156.216
C01189=1045.680,-114.321,-70.329,169.338,32.783,156.216
C01190=1045.686,-114.071,-70.338,169.340,32.783,156.216
C01191=1045.692,-113.822,-70.348,169.343,32.784,156.216
C01192=1045.698,-113.572,-70.357,169.345,32.784,156.216
C01193=1045.704,-113.322,-70.367,169.347,32.784,156.216
C01194=1045.710,-113.072,-70.376,169.350,32.784,156.216
C01195=1045.717,-112.822,-70.386,169.352,32.784,156.216
C01196=1045.723,-112.573,-70.395,169.354,32.784,156.215
C01197=1045.729,-112.323,-70.405,169.357,32.784,156.215
C01198=1045.735,-112.074,-70.415,169.359,32.784,156.215
C01199=1045.742,-111.824,-70.425,169.361,32.785,156.215
C01200=1045.748,-111.574,-70.434,169.364,32.785,156.215
C01201=1045.753,-111.324,-70.445,169.366,32.785,156.215
C01202=1045.759,-111.074,-70.454,169.368,32.785,156.215
C01203=1045.766,-110.824,-70.464,169.371,32.786,156.215
C01204=1045.772,-110.575,-70.473,169.373,32.786,156.215
C01205=1045.778,-110.325,-70.483,169.375,32.786,156.215
C01206=1045.784,-110.075,-70.492,169.377,32.786,156.215
C01207=1045.791,-109.826,-70.503,169.379,32.787,156.215
C01208=1045.797,-109.576,-70.512,169.381,32.786,156.215
C01209=1045.803,-109.326,-70.522,169.384,32.786,156.215
C01210=1045.809,-109.076,-70.531,169.386,32.787,156.215
C01211=1045.815,-108.827,-70.541,169.388,32.787,156.215
C01212=1045.821,-108.576,-70.551,169.391,32.787,156.215
C01213=1045.827,-108.327,-70.561,169.393,32.787,156.214
C01214=1045.833,-108.078,-70.571,169.395,32.788,156.214
C01215=1045.840,-107.828,-70.581,169.398,32.788,156.214
C01216=1045.846,-107.578,-70.590,169.400,32.788,156.214
C01217=1045.852,-107.328,-70.600,169.402,32.788,156.214
C01218=1045.858,-107.079,-70.610,169.405,32.789,156.214
C01219=1045.864,-106.829,-70.620,169.407,32.789,156.214
C01220=1045.870,-106.579,-70.630,169.409,32.789,156.214
C01221=1045.876,-106.330,-70.640,169.412,32.789,156.214
C01222=1045.883,-106.080,-70.650,169.414,32.790,156.214
C01223=1045.888,-105.830,-70.660,169.416,32.790,156.214
C01224=1045.894,-105.580,-70.669,169.419,32.791,156.214
C01225=1045.901,-105.331,-70.680,169.421,32.791,156.214
C01226=1045.907,-105.081,-70.689,169.423,32.791,156.214
C01227=1045.912,-104.831,-70.699,169.426,32.791,156.214
C01228=1045.919,-104.582,-70.710,169.428,32.791,156.214
C01229=1045.925,-104.332,-70.719,169.430,32.792,156.214
C01230=1045.931,-104.082,-70.729,169.432,32.792,156.214
C01231=1045.937,-103.832,-70.740,169.434,32.793,156.214
C01232=1045.944,-103.582,-70.749,169.436,32.793,156.214
C01233=1045.950,-103.333,-70.760,169.439,32.793,156.214
C01234=1045.956,-103.083,-70.770,169.441,32.794,156.214
C01235=1045.962,-102.833,-70.779,169.443,32.794,156.214
C01236=1045.968,-102.584,-70.790,169.446,32.794,156.214
C01237=1045.974,-102.334,-70.800,169.448,32.795,156.214
C01238=1045.980,-102.085,-70.810,169.450,32.795,156.214
C01239=1045.986,-101.835,-70.820,169.452,32.795,156.213
C01240=1045.992,-101.585,-70.829,169.455,32.796,156.213
C01241=1045.999,-101.335,-70.841,169.457,32.796,156.213
C01242=1046.005,-101.085,-70.850,169.459,32.797,156.213
C01243=1046.011,-100.836,-70.860,169.462,32.797,156.213
C01244=1046.017,-100.586,-70.871,169.464,32.797,156.213
C01245=1046.023,-100.337,-70.881,169.466,32.797,156.213
C01246=1046.029,-100.087,-70.890,169.469,32.798,156.213
C01247=1046.036,-99.800,-70.903,169.471,32.798,156.213
C01248=1046.044,-99.513,-70.914,169.474,32.799,156.213
C01249=1046.051,-99.227,-70.926,169.477,32.799,156.213
C01250=1046.058,-98.940,-70.938,169.479,32.799,156.213
C01251=1046.064,-98.690,-70.948,169.482,32.800,156.213
C01252=1046.070,-98.441,-70.958,169.484,32.800,156.213
C01253=1046.076,-98.190,-70.969,169.486,32.801,156.213
C01254=1046.083,-97.941,-70.979,169.488,32.801,156.213
C01255=1046.089,-97.691,-70.989,169.490,32.802,156.213
C01256=1046.095,-97.441,-70.999,169.492,32.802,156.213
C01257=1046.101,-97.192,-71.010,169.494,32.802,156.213
C01258=1046.107,-96.941,-71.020,169.497,32.803,156.213
C01259=1046.114,-96.692,-71.031,169.499,32.803,156.213
C01260=1046.119,-96.442,-71.041,169.501,32.804,156.213
C01261=1046.125,-96.193,-71.052,169.503,32.804,156.213
C01262=1046.131,-95.943,-71.062,169.506,32.805,156.213
C01263=1046.137,-95.693,-71.072,169.508,32.805,156.213
C01264=1046.144,-95.443,-71.083,169.510,32.806,156.213
C01265=1046.150,-95.194,-71.094,169.513,32.807,156.213
C01266=1046.155,-94.944,-71.104,169.515,32.807,156.213
C01267=1046.161,-94.695,-71.114,169.517,32.808,156.213
C01268=1046.168,-94.444,-71.125,169.519,32.808,156.213
C01269=1046.174,-94.195,-71.136,169.522,32.809,156.213
C01270=1046.180,-93.945,-71.146,169.524,32.809,156.213
C01271=1046.185,-93.696,-71.157,169.526,32.810,156.213
C01272=1046.193,-93.446,-71.167,169.528,32.810,156.213
C01273=1046.198,-93.196,-71.177,169.531,32.811,156.213
C01274=1046.204,-92.946,-71.188,169.533,32.811,156.213
C01275=1046.210,-92.697,-71.199,169.535,32.812,156.213
C01276=1046.217,-92.447,-71.210,169.538,32.812,156.213
C01277=1046.223,-92.197,-71.219,169.540,32.813,156.213
C01278=1046.228,-91.948,-71.230,169.542,32.813,156.213
C01279=1046.235,-91.698,-71.241,169.544,32.814,156.213
C01280=1046.241,-91.448,-71.252,169.546,32.814,156.213
C01281=1046.247,-91.199,-71.263,169.548,32.815,156.213
C01282=1046.253,-90.949,-71.273,169.550,32.815,156.213
C01283=1046.259,-90.699,-71.283,169.552,32.816,156.213
C01284=1046.265,-90.449,-71.294,169.555,32.816,156.213
C01285=1046.272,-90.200,-71.305,169.557,32.817,156.213
C01286=1046.277,-89.951,-71.316,169.559,32.818,156.213
C01287=1046.284,-89.700,-71.327,169.561,32.818,156.213
C01288=1046.290,-89.451,-71.337,169.564,32.819,156.213
C01289=1046.296,-89.201,-71.347,169.566,32.819,156.213
C01290=1046.303,-88.951,-71.358,169.568,32.820,156.213
C01291=1046.309,-88.702,-71.369,169.570,32.821,156.213
C01292=1046.314,-88.452,-71.380,169.573,32.821,156.213
C01293=1046.321,-88.202,-71.390,169.575,32.822,156.213
C01294=1046.327,-87.953,-71.401,169.577,32.822,156.213
C01295=1046.333,-87.703,-71.412,169.580,32.823,156.213
C01296=1046.340,-87.453,-71.423,169.582,32.824,156.213
C01297=1046.346,-87.204,-71.434,169.584,32.824,156.213
C01298=1046.352,-86.954,-71.445,169.586,32.825,156.213
C01299=1046.358,-86.705,-71.455,169.589,32.826,156.213
C01300=1046.364,-86.455,-71.466,169.591,32.826,156.213
C01301=1046.371,-86.205,-71.477,169.593,32.827,156.213
C01302=1046.377,-85.956,-71.487,169.595,32.827,156.213
C01303=1046.383,-85.706,-71.499,169.598,32.828,156.213
C01304=1046.389,-85.456,-71.510,169.600,32.829,156.213
C01305=1046.396,-85.207,-71.520,169.601,32.829,156.213
C01306=1046.402,-84.957,-71.531,169.603,32.830,156.213
C01307=1046.408,-84.707,-71.542,169.606,32.831,156.213
C01308=1046.414,-84.457,-71.553,169.608,32.831,156.213
C01309=1046.420,-84.208,-71.564,169.610,32.832,156.213
C01310=1046.427,-83.958,-71.575,169.612,32.832,156.214
C01311=1046.434,-83.673,-71.587,169.615,32.833,156.213
C01312=1046.441,-83.389,-71.599,169.617,32.834,156.214
C01313=1046.448,-83.104,-71.612,169.620,32.834,156.214
C01314=1046.455,-82.820,-71.624,169.623,32.835,156.214
C01315=1046.462,-82.570,-71.635,169.625,32.836,156.214
C01316=1046.468,-82.320,-71.646,169.627,32.836,156.214
C01317=1046.474,-82.070,-71.657,169.629,32.837,156.214
C01318=1046.480,-81.821,-71.668,169.632,32.838,156.214
C01319=1046.486,-81.571,-71.678,169.634,32.838,156.214
C01320=1046.493,-81.322,-71.690,169.636,32.839,156.214
C01321=1046.499,-81.072,-71.701,169.638,32.839,156.214
C01322=1046.505,-80.822,-71.712,169.640,32.840,156.214
C01323=1046.512,-80.572,-71.723,169.643,32.841,156.214
C01324=1046.518,-80.323,-71.734,169.645,32.841,156.214
C01325=1046.524,-80.073,-71.745,169.647,32.842,156.214
C01326=1046.531,-79.824,-71.756,169.649,32.843,156.214
C01327=1046.537,-79.574,-71.767,169.652,32.844,156.214
C01328=1046.543,-79.324,-71.778,169.654,32.844,156.214
C01329=1046.549,-79.074,-71.789,169.656,32.845,156.214
C01330=1046.555,-78.825,-71.800,169.657,32.846,156.214
C01331=1046.562,-78.575,-71.812,169.659,32.847,156.214
C01332=1046.568,-78.326,-71.823,169.662,32.848,156.214
C01333=1046.574,-78.075,-71.834,169.664,32.848,156.214
C01334=1046.580,-77.827,-71.846,169.666,32.849,156.214
C01335=1046.586,-77.576,-71.857,169.668,32.849,156.214
C01336=1046.592,-77.327,-71.868,169.671,32.850,156.214
C01337=1046.598,-77.077,-71.879,169.673,32.851,156.214
C01338=1046.604,-76.828,-71.891,169.675,32.852,156.214
C01339=1046.611,-76.578,-71.902,169.677,32.853,156.215
C01340=1046.616,-76.328,-71.913,169.679,32.854,156.215
C01341=1046.623,-76.079,-71.925,169.682,32.855,156.215
C01342=1046.629,-75.828,-71.936,169.684,32.855,156.215
C01343=1046.635,-75.579,-71.947,169.686,32.856,156.215
C01344=1046.642,-75.329,-71.959,169.688,32.857,156.215
C01345=1046.648,-75.080,-71.970,169.690,32.857,156.215
C01346=1046.654,-74.830,-71.981,169.693,32.858,156.215
C01347=1046.660,-74.581,-71.993,169.695,32.859,156.215
C01348=1046.666,-74.331,-72.004,169.697,32.860,156.215
C01349=1046.673,-74.081,-72.016,169.699,32.861,156.215
C01350=1046.679,-73.831,-72.027,169.701,32.861,156.215
C01351=1046.685,-73.582,-72.039,169.704,32.862,156.215
C01352=1046.691,-73.332,-72.050,169.706,32.863,156.215
C01353=1046.697,-73.082,-72.061,169.708,32.864,156.215
C01354=1046.703,-72.833,-72.073,169.710,32.865,156.215
C01355=1046.709,-72.583,-72.084,169.712,32.866,156.216
C01356=1046.716,-72.333,-72.096,169.714,32.867,156.216
C01357=1046.721,-72.084,-72.107,169.716,32.868,156.216
C01358=1046.727,-71.834,-72.120,169.718,32.869,156.216
C01359=1046.733,-71.584,-72.131,169.720,32.870,156.216
C01360=1046.740,-71.335,-72.143,169.722,32.871,156.216
C01361=1046.746,-71.086,-72.154,169.724,32.871,156.216
C01362=1046.751,-70.835,-72.166,169.726,32.872,156.216
C01363=1046.758,-70.586,-72.178,169.729,32.874,156.216
C01364=1046.764,-70.336,-72.189,169.731,32.875,156.216
C01365=1046.770,-70.087,-72.201,169.733,32.875,156.216
C01366=1046.776,-69.836,-72.213,169.735,32.876,156.216
C01367=1046.782,-69.587,-72.224,169.737,32.877,156.216
C01368=1046.788,-69.337,-72.236,169.739,32.878,156.217
C01369=1046.794,-69.088,-72.247,169.741,32.879,156.217
C01370=1046.800,-68.838,-72.260,169.744,32.880,156.217
C01371=1046.807,-68.588,-72.271,169.746,32.881,156.217
C01372=1046.813,-68.339,-72.283,169.748,32.882,156.217
C01373=1046.819,-68.090,-72.294,169.750,32.883,156.217
C01374=1046.825,-67.839,-72.306,169.752,32.884,156.217
C01375=1046.832,-67.557,-72.320,169.755,32.885,156.217
C01376=1046.839,-67.275,-72.333,169.757,32.886,156.217
C01377=1046.847,-66.993,-72.346,169.760,32.887,156.217
C01378=1046.853,-66.710,-72.359,169.762,32.888,156.217
C01379=1046.859,-66.461,-72.371,169.764,32.889,156.218
C01380=1046.865,-66.211,-72.383,169.766,32.890,156.218
C01381=1046.872,-65.961,-72.395,169.768,32.891,156.218
C01382=1046.878,-65.711,-72.407,169.771,32.892,156.218
C01383=1046.884,-65.463,-72.419,169.773,32.893,156.218
C01384=1046.890,-65.212,-72.430,169.774,32.894,156.218
C01385=1046.897,-64.963,-72.442,169.776,32.895,156.218
C01386=1046.902,-64.714,-72.454,169.778,32.896,156.218
C01387=1046.908,-64.464,-72.466,169.780,32.896,156.218
C01388=1046.915,-64.214,-72.477,169.782,32.898,156.218
C01389=1046.921,-63.964,-72.490,169.785,32.899,156.218
C01390=1046.927,-63.715,-72.501,169.787,32.900,156.218
C01391=1046.933,-63.465,-72.513,169.789,32.900,156.219
C01392=1046.939,-63.215,-72.525,169.791,32.902,156.219
C01393=1046.946,-62.965,-72.537,169.793,32.903,156.219
C01394=1046.952,-62.717,-72.549,169.795,32.904,156.219
C01395=1046.958,-62.467,-72.561,169.797,32.904,156.219
C01396=1046.964,-62.217,-72.573,169.800,32.906,156.219
C01397=1046.971,-61.968,-72.585,169.802,32.907,156.219
C01398=1046.977,-61.717,-72.597,169.804,32.908,156.219
C01399=1046.983,-61.468,-72.609,169.806,32.908,156.219
C01400=1046.989,-61.219,-72.621,169.808,32.910,156.219
C01401=1046.995,-60.969,-72.633,169.810,32.911,156.220
C01402=1047.002,-60.719,-72.645,169.812,32.912,156.220
C01403=1047.008,-60.470,-72.657,169.815,32.912,156.220
C01404=1047.014,-60.220,-72.670,169.817,32.914,156.220
C01405=1047.020,-59.970,-72.681,169.819,32.915,156.220
C01406=1047.027,-59.721,-72.692,169.821,32.916,156.220
C01407=1047.033,-59.471,-72.705,169.823,32.916,156.220
C01408=1047.039,-59.221,-72.717,169.825,32.918,156.220
C01409=1047.046,-58.972,-72.729,169.827,32.919,156.220
C01410=1047.052,-58.722,-72.742,169.829,32.919,156.220
C01411=1047.058,-58.473,-72.753,169.832,32.921,156.221
C01412=1047.065,-58.223,-72.765,169.834,32.922,156.221
C01413=1047.070,-57.973,-72.778,169.835,32.923,156.221
C01414=1047.077,-57.724,-72.790,169.837,32.923,156.221
C01415=1047.083,-57.474,-72.802,169.839,32.925,156.221
C01416=1047.090,-57.224,-72.814,169.841,32.926,156.221
C01417=1047.096,-56.975,-72.826,169.843,32.927,156.221
C01418=1047.102,-56.725,-72.839,169.845,32.928,156.221
C01419=1047.109,-56.475,-72.851,169.848,32.929,156.221
C01420=1047.115,-56.226,-72.863,169.850,32.930,156.221
C01421=1047.121,-55.977,-72.875,169.852,32.931,156.222
C01422=1047.127,-55.727,-72.887,169.854,32.932,156.222
C01423=1047.133,-55.477,-72.899,169.856,32.933,156.222
C01424=1047.140,-55.228,-72.911,169.858,32.934,156.222
C01425=1047.147,-54.978,-72.923,169.860,32.935,156.222
C01426=1047.153,-54.728,-72.936,169.862,32.936,156.222
C01427=1047.159,-54.478,-72.948,169.864,32.937,156.222
C01428=1047.165,-54.229,-72.960,169.867,32.938,156.222
C01429=1047.172,-53.979,-72.972,169.869,32.939,156.222
C01430=1047.179,-53.730,-72.985,169.871,32.941,156.222
C01431=1047.185,-53.480,-72.997,169.873,32.941,156.223
C01432=1047.191,-53.231,-73.009,169.875,32.942,156.223
C01433=1047.197,-52.981,-73.022,169.877,32.944,156.223
C01434=1047.204,-52.731,-73.034,169.879,32.944,156.223
C01435=1047.210,-52.482,-73.046,169.881,32.945,156.223
C01436=1047.216,-52.232,-73.058,169.883,32.947,156.223
C01437=1047.223,-51.982,-73.070,169.885,32.948,156.223
C01438=1047.229,-51.733,-73.084,169.888,32.948,156.223
C01439=1047.236,-51.452,-73.096,169.890,32.950,156.223
C01440=1047.244,-51.170,-73.111,169.892,32.951,156.224
C01441=1047.251,-50.890,-73.125,169.895,32.952,156.224
C01442=1047.259,-50.609,-73.139,169.896,32.954,156.224
C01443=1047.265,-50.359,-73.151,169.898,32.955,156.224
C01444=1047.270,-50.109,-73.164,169.900,32.956,156.224
C01445=1047.277,-49.860,-73.176,169.902,32.957,156.224
C01446=1047.283,-49.610,-73.189,169.904,32.958,156.224
C01447=1047.289,-49.360,-73.202,169.906,32.959,156.224
C01448=1047.295,-49.110,-73.214,169.908,32.961,156.225
C01449=1047.302,-48.861,-73.227,169.910,32.962,156.225
C01450=1047.308,-48.611,-73.239,169.913,32.963,156.225
C01451=1047.314,-48.362,-73.252,169.915,32.964,156.225
C01452=1047.320,-48.112,-73.265,169.917,32.966,156.225
C01453=1047.327,-47.863,-73.277,169.919,32.967,156.225
C01454=1047.333,-47.613,-73.290,169.921,32.968,156.225
C01455=1047.339,-47.364,-73.303,169.923,32.969,156.226
C01456=1047.345,-47.114,-73.316,169.925,32.970,156.226
C01457=1047.351,-46.864,-73.327,169.927,32.972,156.226
C01458=1047.358,-46.615,-73.341,169.929,32.973,156.226
C01459=1047.364,-46.365,-73.353,169.931,32.974,156.226
C01460=1047.370,-46.116,-73.367,169.933,32.975,156.226
C01461=1047.376,-45.866,-73.379,169.935,32.976,156.226
C01462=1047.382,-45.616,-73.391,169.937,32.978,156.227
C01463=1047.389,-45.367,-73.404,169.939,32.979,156.227
C01464=1047.394,-45.117,-73.417,169.941,32.980,156.227
C01465=1047.401,-44.868,-73.430,169.943,32.981,156.227
C01466=1047.407,-44.618,-73.442,169.945,32.982,156.227
C01467=1047.413,-44.368,-73.455,169.947,32.984,156.227
C01468=1047.419,-44.119,-73.468,169.949,32.985,156.227
C01469=1047.425,-43.869,-73.481,169.951,32.986,156.228
C01470=1047.432,-43.619,-73.494,169.954,32.987,156.228
C01471=1047.439,-43.370,-73.506,169.956,32.989,156.228
C01472=1047.445,-43.120,-73.519,169.958,32.990,156.228
C01473=1047.451,-42.871,-73.532,169.960,32.991,156.228
C01474=1047.457,-42.621,-73.545,169.962,32.993,156.228
C01475=1047.463,-42.371,-73.558,169.964,32.993,156.228
C01476=1047.470,-42.122,-73.570,169.965,32.995,156.229
C01477=1047.476,-41.873,-73.583,169.967,32.996,156.229
C01478=1047.483,-41.623,-73.597,169.969,32.997,156.229
C01479=1047.489,-41.373,-73.609,169.971,32.999,156.229
C01480=1047.495,-41.123,-73.622,169.973,33.000,156.229
C01481=1047.501,-40.874,-73.636,169.975,33.001,156.229
C01482=1047.508,-40.625,-73.648,169.977,33.002,156.229
C01483=1047.514,-40.375,-73.661,169.979,33.004,156.230
C01484=1047.520,-40.125,-73.673,169.981,33.005,156.230
C01485=1047.527,-39.875,-73.687,169.983,33.006,156.230
C01486=1047.533,-39.626,-73.700,169.985,33.007,156.230
C01487=1047.539,-39.376,-73.713,169.987,33.008,156.230
C01488=1047.546,-39.127,-73.726,169.989,33.010,156.230
C01489=1047.552,-38.878,-73.738,169.991,33.011,156.230
C01490=1047.558,-38.628,-73.752,169.993,33.013,156.231
C01491=1047.565,-38.378,-73.765,169.995,33.013,156.231
C01492=1047.571,-38.128,-73.778,169.997,33.015,156.231
C01493=1047.577,-37.879,-73.791,169.999,33.016,156.231
C01494=1047.583,-37.630,-73.804,170.001,33.018,156.231
C01495=1047.589,-37.380,-73.817,170.003,33.019,156.231
C01496=1047.595,-37.131,-73.830,170.005,33.021,156.232
C01497=1047.602,-36.881,-73.844,170.007,33.021,156.232
C01498=1047.608,-36.632,-73.857,170.009,33.023,156.232
C01499=1047.613,-36.381,-73.870,170.011,33.024,156.232
C01500=1047.620,-36.132,-73.883,170.013,33.026,156.232
C01501=1047.626,-35.883,-73.897,170.015,33.027,156.232
C01502=1047.633,-35.633,-73.910,170.017,33.029,156.233
C01503=1047.639,-35.352,-73.924,170.019,33.030,156.233
C01504=1047.646,-35.072,-73.939,170.022,33.032,156.233
C01505=1047.653,-34.791,-73.955,170.024,33.033,156.233
C01506=1047.660,-34.510,-73.969,170.026,33.034,156.233
C01507=1047.666,-34.261,-73.982,170.028,33.036,156.234
C01508=1047.673,-34.011,-73.996,170.030,33.037,156.234
C01509=1047.679,-33.762,-74.009,170.032,33.039,156.234
C01510=1047.686,-33.512,-74.022,170.034,33.040,156.234
C01511=1047.692,-33.263,-74.036,170.036,33.041,156.234
C01512=1047.698,-33.013,-74.048,170.037,33.042,156.234
C01513=1047.704,-32.763,-74.062,170.039,33.044,156.235
C01514=1047.710,-32.514,-74.076,170.041,33.045,156.235
C01515=1047.716,-32.265,-74.089,170.043,33.047,156.235
C01516=1047.723,-32.015,-74.103,170.045,33.048,156.235
C01517=1047.729,-31.765,-74.116,170.047,33.050,156.235
C01518=1047.735,-31.516,-74.129,170.049,33.051,156.235
C01519=1047.742,-31.267,-74.142,170.051,33.052,156.236
C01520=1047.748,-31.016,-74.155,170.053,33.053,156.236
C01521=1047.754,-30.767,-74.169,170.055,33.055,156.236
C01522=1047.761,-30.518,-74.182,170.057,33.056,156.236
C01523=1047.767,-30.268,-74.195,170.059,33.058,156.236
C01524=1047.773,-30.018,-74.209,170.061,33.059,156.236
C01525=1047.779,-29.769,-74.223,170.063,33.060,156.237
C01526=1047.786,-29.519,-74.236,170.065,33.062,156.237
C01527=1047.792,-29.270,-74.249,170.066,33.063,156.237
C01528=1047.798,-29.020,-74.263,170.068,33.065,156.237
C01529=1047.805,-28.770,-74.276,170.070,33.065,156.237
C01530=1047.811,-28.521,-74.290,170.072,33.067,156.237
C01531=1047.818,-28.272,-74.303,170.074,33.068,156.238
C01532=1047.824,-28.022,-74.317,170.076,33.070,156.238
C01533=1047.830,-27.772,-74.330,170.078,33.071,156.238
C01534=1047.836,-27.523,-74.344,170.080,33.073,156.238
C01535=1047.843,-27.273,-74.357,170.082,33.074,156.238
C01536=1047.849,-27.024,-74.371,170.084,33.076,156.239
C01537=1047.856,-26.774,-74.384,170.086,33.077,156.239
C01538=1047.861,-26.524,-74.398,170.088,33.078,156.239
C01539=1047.868,-26.275,-74.411,170.090,33.080,156.239
C01540=1047.874,-26.025,-74.425,170.092,33.081,156.239
C01541=1047.880,-25.775,-74.439,170.094,33.083,156.240
C01542=1047.886,-25.526,-74.452,170.096,33.084,156.240
C01543=1047.892,-25.277,-74.467,170.098,33.086,156.240
C01544=1047.899,-25.027,-74.480,170.100,33.087,156.240
C01545=1047.905,-24.778,-74.494,170.102,33.088,156.240
C01546=1047.911,-24.528,-74.508,170.103,33.090,156.241
C01547=1047.917,-24.278,-74.521,170.105,33.092,156.241
C01548=1047.923,-24.029,-74.534,170.107,33.093,156.241
C01549=1047.930,-23.780,-74.549,170.109,33.095,156.241
C01550=1047.936,-23.530,-74.563,170.111,33.096,156.241
C01551=1047.942,-23.280,-74.577,170.113,33.098,156.241
C01552=1047.948,-23.031,-74.590,170.115,33.099,156.242
C01553=1047.955,-22.781,-74.603,170.117,33.100,156.242
C01554=1047.961,-22.531,-74.618,170.119,33.102,156.242
C01555=1047.967,-22.283,-74.632,170.121,33.103,156.242
C01556=1047.973,-22.032,-74.646,170.123,33.105,156.242
C01557=1047.979,-21.783,-74.659,170.124,33.106,156.243
C01558=1047.986,-21.534,-74.672,170.126,33.108,156.243
C01559=1047.992,-21.284,-74.687,170.127,33.110,156.243
C01560=1047.998,-21.035,-74.701,170.129,33.111,156.243
C01561=1048.005,-20.785,-74.714,170.131,33.112,156.243
C01562=1048.010,-20.535,-74.728,170.133,33.114,156.244
C01563=1048.018,-20.286,-74.742,170.135,33.115,156.244
C01564=1048.023,-20.036,-74.756,170.137,33.117,156.244
C01565=1048.030,-19.786,-74.770,170.139,33.118,156.244
C01566=1048.036,-19.537,-74.785,170.141,33.120,156.244
C01567=1048.043,-19.256,-74.799,170.143,33.122,156.245
C01568=1048.051,-18.974,-74.815,170.145,33.123,156.245
C01569=1048.057,-18.693,-74.831,170.147,33.124,156.245
C01570=1048.064,-18.412,-74.847,170.149,33.126,156.245
C01571=1048.070,-18.162,-74.861,170.151,33.128,156.246
C01572=1048.077,-17.913,-74.875,170.153,33.129,156.246
C01573=1048.083,-17.663,-74.889,170.155,33.131,156.246
C01574=1048.089,-17.414,-74.902,170.157,33.132,156.246
C01575=1048.096,-17.164,-74.917,170.159,33.134,156.246
C01576=1048.102,-16.915,-74.930,170.161,33.135,156.247
C01577=1048.109,-16.665,-74.945,170.163,33.137,156.247
C01578=1048.115,-16.416,-74.959,170.165,33.139,156.247
C01579=1048.121,-16.166,-74.972,170.167,33.140,156.247
C01580=1048.128,-15.916,-74.987,170.169,33.141,156.247
C01581=1048.134,-15.667,-75.001,170.170,33.143,156.248
C01582=1048.140,-15.417,-75.015,170.172,33.144,156.248
C01583=1048.147,-15.168,-75.029,170.174,33.146,156.248
C01584=1048.153,-14.918,-75.044,170.176,33.148,156.248
C01585=1048.159,-14.669,-75.057,170.178,33.149,156.248
C01586=1048.165,-14.419,-75.071,170.180,33.150,156.249
C01587=1048.171,-14.170,-75.086,170.182,33.152,156.249
C01588=1048.178,-13.920,-75.099,170.184,33.154,156.249
C01589=1048.184,-13.671,-75.114,170.185,33.155,156.249
C01590=1048.190,-13.421,-75.129,170.187,33.157,156.249
C01591=1048.196,-13.172,-75.142,170.189,33.158,156.250
C01592=1048.203,-12.922,-75.157,170.191,33.160,156.250
C01593=1048.209,-12.672,-75.171,170.193,33.162,156.250
C01594=1048.215,-12.423,-75.185,170.195,33.163,156.250
C01595=1048.221,-12.173,-75.200,170.197,33.164,156.251
C01596=1048.227,-11.924,-75.214,170.198,33.166,156.251
C01597=1048.234,-11.674,-75.228,170.200,33.168,156.251
C01598=1048.240,-11.425,-75.242,170.202,33.169,156.251
C01599=1048.246,-11.176,-75.257,170.204,33.171,156.252
C01600=1048.252,-10.926,-75.271,170.206,33.173,156.252
C01601=1048.259,-10.677,-75.286,170.208,33.174,156.252
C01602=1048.265,-10.426,-75.300,170.210,33.176,156.252
C01603=1048.270,-10.177,-75.314,170.212,33.178,156.252
C01604=1048.278,-9.928,-75.329,170.213,33.179,156.253
C01605=1048.283,-9.678,-75.343,170.215,33.180,156.253
C01606=1048.289,-9.429,-75.358,170.217,33.182,156.253
C01607=1048.297,-9.179,-75.372,170.219,33.184,156.253
C01608=1048.302,-8.930,-75.386,170.221,33.185,156.253
C01609=1048.308,-8.680,-75.401,170.223,33.187,156.254
C01610=1048.316,-8.431,-75.415,170.224,33.189,156.254
C01611=1048.321,-8.181,-75.429,170.226,33.190,156.254
C01612=1048.327,-7.932,-75.444,170.228,33.192,156.254
C01613=1048.334,-7.682,-75.459,170.230,33.193,156.255
C01614=1048.340,-7.433,-75.472,170.232,33.195,156.255
C01615=1048.346,-7.183,-75.487,170.234,33.196,156.255
C01616=1048.353,-6.933,-75.502,170.236,33.198,156.255
C01617=1048.359,-6.684,-75.517,170.237,33.200,156.256
C01618=1048.365,-6.434,-75.530,170.239,33.201,156.256
C01619=1048.372,-6.185,-75.545,170.241,33.203,156.256
C01620=1048.378,-5.936,-75.560,170.242,33.204,156.256
C01621=1048.385,-5.687,-75.574,170.244,33.206,156.256
C01622=1048.391,-5.436,-75.588,170.246,33.208,156.257
C01623=1048.396,-5.187,-75.603,170.248,33.209,156.257
C01624=1048.403,-4.938,-75.618,170.249,33.211,156.257
C01625=1048.410,-4.688,-75.632,170.251,33.212,156.257
C01626=1048.416,-4.439,-75.647,170.253,33.214,156.257
C01627=1048.422,-4.189,-75.661,170.255,33.215,156.258
C01628=1048.428,-3.939,-75.676,170.257,33.217,156.258
C01629=1048.435,-3.690,-75.690,170.259,33.219,156.258
C01630=1048.441,-3.441,-75.705,170.260,33.220,156.258
C01631=1048.448,-3.158,-75.721,170.262,33.222,156.259
C01632=1048.456,-2.875,-75.738,170.264,33.224,156.259
C01633=1048.462,-2.592,-75.756,170.267,33.226,156.259
C01634=1048.469,-2.309,-75.772,170.269,33.228,156.260
C01635=1048.475,-2.059,-75.787,170.270,33.230,156.260
C01636=1048.481,-1.810,-75.802,170.272,33.231,156.260
C01637=1048.487,-1.561,-75.816,170.274,33.233,156.260
C01638=1048.494,-1.311,-75.831,170.276,33.234,156.260
C01639=1048.500,-1.061,-75.846,170.278,33.236,156.261
C01640=1048.506,-0.812,-75.861,170.279,33.238,156.261
C01641=1048.512,-0.563,-75.876,170.281,33.240,156.261
C01642=1048.519,-0.313,-75.891,170.283,33.241,156.261
C01643=1048.525,-0.063,-75.906,170.285,33.243,156.262
C01644=1048.531,0.186,-75.920,170.287,33.245,156.262
C01645=1048.537,0.435,-75.935,170.288,33.247,156.262
C01646=1048.544,0.685,-75.950,170.290,33.248,156.262
C01647=1048.549,0.934,-75.965,170.292,33.250,156.263
C01648=1048.556,1.184,-75.980,170.294,33.252,156.263
C01649=1048.561,1.434,-75.995,170.296,33.254,156.263
C01650=1048.568,1.683,-76.010,170.297,33.255,156.263
C01651=1048.574,1.932,-76.025,170.299,33.257,156.264
C01652=1048.580,2.182,-76.040,170.301,33.258,156.264
C01653=1048.586,2.431,-76.055,170.303,33.260,156.264
C01654=1048.593,2.681,-76.070,170.305,33.262,156.264
C01655=1048.599,2.931,-76.085,170.306,33.264,156.265
C01656=1048.605,3.180,-76.099,170.308,33.265,156.265
C01657=1048.611,3.429,-76.114,170.310,33.267,156.265
C01658=1048.618,3.679,-76.129,170.312,33.269,156.265
C01659=1048.624,3.928,-76.145,170.313,33.271,156.266
C01660=1048.631,4.178,-76.160,170.315,33.272,156.266
C01661=1048.636,4.427,-76.174,170.317,33.274,156.266
C01662=1048.642,4.677,-76.190,170.319,33.275,156.266
C01663=1048.648,4.926,-76.205,170.321,33.277,156.267
C01664=1048.655,5.176,-76.220,170.322,33.279,156.267
C01665=1048.661,5.426,-76.235,170.324,33.280,156.267
C01666=1048.667,5.674,-76.250,170.326,33.282,156.267
C01667=1048.674,5.924,-76.265,170.328,33.284,156.268
C01668=1048.680,6.173,-76.280,170.330,33.286,156.268
C01669=1048.686,6.423,-76.295,170.331,33.287,156.268
C01670=1048.693,6.673,-76.310,170.333,33.289,156.268
C01671=1048.700,6.922,-76.325,170.335,33.290,156.269
C01672=1048.705,7.172,-76.341,170.337,33.292,156.269
C01673=1048.711,7.421,-76.355,170.338,33.294,156.269
C01674=1048.717,7.670,-76.370,170.340,33.296,156.269
C01675=1048.724,7.920,-76.385,170.342,33.297,156.270
C01676=1048.730,8.169,-76.401,170.344,33.299,156.270
C01677=1048.737,8.419,-76.416,170.346,33.301,156.270
C01678=1048.743,8.668,-76.431,170.347,33.303,156.270
C01679=1048.750,8.918,-76.446,170.349,33.304,156.271
C01680=1048.756,9.167,-76.462,170.351,33.306,156.271
C01681=1048.762,9.417,-76.477,170.353,33.308,156.271
C01682=1048.768,9.666,-76.492,170.354,33.309,156.271
C01683=1048.774,9.915,-76.507,170.356,33.311,156.272
C01684=1048.781,10.165,-76.522,170.358,33.313,156.272
C01685=1048.787,10.414,-76.537,170.360,33.314,156.272
C01686=1048.794,10.664,-76.552,170.361,33.316,156.272
C01687=1048.800,10.913,-76.568,170.363,33.318,156.273
C01688=1048.806,11.163,-76.583,170.365,33.320,156.273
C01689=1048.812,11.413,-76.598,170.367,33.321,156.273
C01690=1048.819,11.662,-76.614,170.369,33.323,156.273
C01691=1048.825,11.911,-76.629,170.370,33.324,156.274
C01692=1048.832,12.161,-76.644,170.372,33.326,156.274
C01693=1048.838,12.410,-76.659,170.374,33.328,156.274
C01694=1048.844,12.660,-76.675,170.376,33.330,156.274
C01695=1048.851,12.944,-76.692,170.378,33.331,156.275
C01696=1048.859,13.229,-76.709,170.380,33.333,156.275
C01697=1048.866,13.514,-76.727,170.382,33.335,156.275
C01698=1048.874,13.799,-76.744,170.384,33.337,156.276
C01699=1048.880,14.048,-76.761,170.385,33.339,156.276
C01700=1048.886,14.298,-76.776,170.387,33.341,156.276
C01701=1048.892,14.548,-76.791,170.389,33.343,156.276
C01702=1048.898,14.797,-76.807,170.391,33.344,156.277
C01703=1048.905,15.047,-76.822,170.392,33.346,156.277
C01704=1048.911,15.296,-76.837,170.394,33.348,156.277
C01705=1048.917,15.546,-76.853,170.396,33.350,156.277
C01706=1048.924,15.795,-76.869,170.398,33.352,156.278
C01707=1048.929,16.045,-76.884,170.399,33.353,156.278
C01708=1048.936,16.294,-76.900,170.401,33.355,156.278
C01709=1048.943,16.543,-76.915,170.403,33.357,156.279
C01710=1048.948,16.793,-76.931,170.405,33.358,156.279
C01711=1048.955,17.042,-76.947,170.406,33.360,156.279
C01712=1048.961,17.292,-76.962,170.408,33.362,156.279
C01713=1048.967,17.541,-76.978,170.410,33.364,156.280
C01714=1048.974,17.790,-76.993,170.411,33.366,156.280
C01715=1048.980,18.040,-77.009,170.413,33.367,156.280
C01716=1048.986,18.289,-77.024,170.415,33.369,156.280
C01717=1048.992,18.539,-77.040,170.417,33.371,156.281
C01718=1048.999,18.788,-77.056,170.418,33.373,156.281
C01719=1049.005,19.037,-77.071,170.420,33.375,156.281
C01720=1049.011,19.287,-77.087,170.422,33.376,156.281
C01721=1049.018,19.536,-77.102,170.424,33.378,156.282
C01722=1049.024,19.786,-77.118,170.425,33.380,156.282
C01723=1049.030,20.035,-77.134,170.427,33.381,156.282
C01724=1049.036,20.285,-77.150,170.429,33.383,156.283
C01725=1049.043,20.534,-77.165,170.430,33.385,156.283
C01726=1049.048,20.783,-77.181,170.432,33.387,156.283
C01727=1049.055,21.033,-77.196,170.434,33.389,156.283
C01728=1049.061,21.282,-77.213,170.436,33.391,156.284
C01729=1049.068,21.531,-77.228,170.437,33.392,156.284
C01730=1049.073,21.781,-77.244,170.439,33.394,156.284
C01731=1049.079,22.031,-77.260,170.441,33.396,156.284
C01732=1049.086,22.280,-77.276,170.442,33.397,156.285
C01733=1049.092,22.529,-77.292,170.444,33.399,156.285
C01734=1049.098,22.779,-77.307,170.446,33.401,156.285
C01735=1049.104,23.028,-77.323,170.448,33.403,156.286
C01736=1049.111,23.278,-77.339,170.449,33.405,156.286
C01737=1049.117,23.527,-77.356,170.451,33.407,156.286
C01738=1049.124,23.777,-77.371,170.453,33.409,156.286
C01739=1049.130,24.026,-77.387,170.454,33.410,156.287
C01740=1049.136,24.275,-77.403,170.456,33.412,156.287
C01741=1049.142,24.524,-77.419,170.458,33.414,156.287
C01742=1049.148,24.774,-77.435,170.460,33.416,156.287
C01743=1049.155,25.023,-77.450,170.461,33.418,156.288
C01744=1049.161,25.273,-77.466,170.463,33.420,156.288
C01745=1049.167,25.522,-77.482,170.465,33.421,156.288
C01746=1049.174,25.772,-77.498,170.466,33.423,156.289
C01747=1049.179,25.995,-77.513,170.468,33.424,156.289
C01748=1049.185,26.219,-77.527,170.469,33.426,156.289
C01749=1049.190,26.442,-77.541,170.471,33.428,156.289
C01750=1049.196,26.665,-77.556,170.473,33.430,156.290
C01751=1049.201,26.889,-77.570,170.474,33.431,156.290
C01752=1049.207,27.112,-77.583,170.476,33.433,156.290
C01753=1049.213,27.336,-77.598,170.477,33.434,156.290
C01754=1049.219,27.559,-77.613,170.479,33.436,156.291
C01755=1049.225,27.809,-77.629,170.480,33.438,156.291
C01756=1049.231,28.058,-77.645,170.482,33.440,156.291
C01757=1049.237,28.307,-77.661,170.484,33.441,156.291
C01758=1049.243,28.556,-77.677,170.485,33.443,156.292
C01759=1049.252,28.895,-77.699,170.488,33.446,156.292
C01760=1049.261,29.233,-77.721,170.490,33.448,156.293
C01761=1049.269,29.572,-77.743,170.492,33.451,156.293
C01762=1049.277,29.909,-77.764,170.495,33.453,156.293
C01763=1049.283,30.158,-77.781,170.496,33.455,156.294
C01764=1049.290,30.408,-77.797,170.498,33.457,156.294
C01765=1049.296,30.658,-77.813,170.500,33.459,156.294
C01766=1049.302,30.907,-77.830,170.501,33.460,156.294
C01767=1049.308,31.156,-77.845,170.503,33.462,156.295
C01768=1049.314,31.405,-77.862,170.505,33.464,156.295
C01769=1049.321,31.656,-77.878,170.506,33.466,156.295
C01770=1049.327,31.905,-77.894,170.508,33.468,156.296
C01771=1049.333,32.154,-77.911,170.510,33.470,156.296
C01772=1049.339,32.403,-77.926,170.511,33.472,156.296
C01773=1049.345,32.653,-77.943,170.513,33.474,156.296
C01774=1049.351,32.902,-77.959,170.515,33.476,156.297
C01775=1049.358,33.152,-77.976,170.516,33.477,156.297
C01776=1049.364,33.401,-77.992,170.518,33.479,156.297
C01777=1049.371,33.650,-78.008,170.521,33.481,156.298
C01778=1049.377,33.899,-78.024,170.522,33.483,156.298
C01779=1049.383,34.149,-78.041,170.524,33.485,156.298
C01780=1049.389,34.399,-78.057,170.526,33.486,156.298
C01781=1049.395,34.648,-78.074,170.528,33.488,156.299
C01782=1049.401,34.897,-78.090,170.529,33.490,156.299
C01783=1049.408,35.147,-78.106,170.531,33.492,156.299
C01784=1049.414,35.396,-78.122,170.533,33.494,156.300
C01785=1049.421,35.645,-78.139,170.534,33.496,156.300
C01786=1049.427,35.894,-78.155,170.536,33.498,156.300
C01787=1049.433,36.144,-78.172,170.538,33.500,156.300
C01788=1049.439,36.394,-78.188,170.539,33.501,156.301
C01789=1049.446,36.643,-78.204,170.541,33.503,156.301
C01790=1049.452,36.892,-78.221,170.543,33.505,156.301
C01791=1049.459,37.142,-78.237,170.544,33.507,156.302
C01792=1049.465,37.391,-78.254,170.546,33.509,156.302
C01793=1049.470,37.640,-78.270,170.548,33.510,156.302
C01794=1049.477,37.890,-78.287,170.549,33.512,156.302
C01795=1049.483,38.139,-78.304,170.551,33.514,156.303
C01796=1049.489,38.388,-78.320,170.553,33.516,156.303
C01797=1049.495,38.638,-78.336,170.554,33.518,156.303
C01798=1049.502,38.888,-78.353,170.556,33.520,156.304
C01799=1049.508,39.137,-78.370,170.558,33.522,156.304
C01800=1049.514,39.386,-78.386,170.559,33.524,156.304
C01801=1049.520,39.635,-78.402,170.561,33.526,156.305
C01802=1049.527,39.885,-78.420,170.563,33.528,156.305
C01803=1049.533,40.134,-78.436,170.564,33.530,156.305
C01804=1049.539,40.383,-78.452,170.566,33.532,156.306
C01805=1049.545,40.633,-78.469,170.568,33.534,156.306
C01806=1049.551,40.882,-78.486,170.569,33.536,156.306
C01807=1049.557,41.132,-78.502,170.571,33.537,156.306
C01808=1049.564,41.381,-78.520,170.573,33.539,156.307
C01809=1049.569,41.631,-78.536,170.574,33.541,156.307
C01810=1049.576,41.879,-78.553,170.576,33.543,156.307
C01811=1049.582,42.129,-78.570,170.577,33.545,156.308
C01812=1049.588,42.379,-78.586,170.579,33.547,156.308
C01813=1049.594,42.627,-78.603,170.581,33.549,156.308
C01814=1049.601,42.878,-78.620,170.582,33.550,156.308
C01815=1049.607,43.127,-78.636,170.584,33.552,156.309
C01816=1049.613,43.376,-78.653,170.586,33.554,156.309
C01817=1049.620,43.626,-78.669,170.587,33.556,156.309
C01818=1049.625,43.875,-78.687,170.589,33.558,156.310
